LIN {X 0,Y 247.028,Z 622.984,A -85,B 0,C 180,E1 -18810.001,E2 -18810.001} C_VEL
LIN {X 0,Y 246.912,Z 622.365,A -85,B 0,C 180,E1 -18813.264,E2 -18813.264} C_VEL
LIN {X 0,Y 246.95,Z 620.585,A -85,B 0,C 180,E1 -18816.537,E2 -18816.537} C_VEL
LIN {X 0,Y 247.222,Z 617.621,A -85,B 0,C 180,E1 -18819.822,E2 -18819.822} C_VEL
LIN {X 0,Y 248.048,Z 613.414,A -85,B 0,C 180,E1 -18823.102,E2 -18823.102} C_VEL
LIN {X 0,Y 249.417,Z 607.853,A -85,B 0,C 180,E1 -18826.367,E2 -18826.367} C_VEL
LIN {X 0,Y 251.498,Z 600.794,A -85,B 0,C 180,E1 -18829.594,E2 -18829.594} C_VEL
LIN {X 0,Y 253.864,Z 593.254,A -85,B 0,C 180,E1 -18832.375,E2 -18832.375} C_VEL
LIN {X 0,Y 256.688,Z 584.514,A -85,B 0,C 180,E1 -18835.005,E2 -18835.005} C_VEL
LIN {X 0,Y 259.73,Z 574.915,A -85,B 0,C 180,E1 -18837.388,E2 -18837.388} C_VEL
LIN {X 0,Y 263.123,Z 564.018,A -85,B 0,C 180,E1 -18839.614,E2 -18839.614} C_VEL
LIN {X 0,Y 266.592,Z 552.132,A -85,B 0,C 180,E1 -18841.599,E2 -18841.599} C_VEL
LIN {X 0,Y 270.114,Z 539.053,A -85,B 0,C 180,E1 -18843.357,E2 -18843.357} C_VEL
LIN {X 0,Y 273.369,Z 524.786,A -85,B 0,C 180,E1 -18844.892,E2 -18844.892} C_VEL
LIN {X 0,Y 276.063,Z 510.769,A -85,B 0,C 180,E1 -18846.067,E2 -18846.067} C_VEL
LIN {X 0,Y 278.527,Z 495.775,A -85,B 0,C 180,E1 -18846.989,E2 -18846.989} C_VEL
LIN {X 0,Y 280.288,Z 480.084,A -85,B 0,C 180,E1 -18847.676,E2 -18847.676} C_VEL
LIN {X 0,Y 281.51,Z 460.198,A -85,B 0,C 180,E1 -18848.22,E2 -18848.22} C_VEL
LIN {X 0,Y 285.491,Z 375.925,A -85,B 0,C 180,E1 -18850.259,E2 -18850.259} C_VEL
LIN {X 0,Y 284.689,Z 371.253,A -85,B 0,C 180,E1 -18850.546,E2 -18850.546} C_VEL
LIN {X 0,Y 277.977,Z 355.557,A -85,B 0,C 180,E1 -18852.259,E2 -18852.259} C_VEL
LIN {X 0,Y 269.371,Z 338.427,A -85,B 0,C 180,E1 -18854.55,E2 -18854.55} C_VEL
LIN {X 0,Y 262.911,Z 327.193,A -85,B 0,C 180,E1 -18856.37,E2 -18856.37} C_VEL
LIN {X 0,Y 257.461,Z 318.292,A -85,B 0,C 180,E1 -18858.004,E2 -18858.004} C_VEL
LIN {X 0,Y 253.878,Z 312.814,A -85,B 0,C 180,E1 -18859.131,E2 -18859.131} C_VEL
LIN {X 0,Y 251.04,Z 308.21,A -85,B 0,C 180,E1 -18860.113,E2 -18860.113} C_VEL
LIN {X 0,Y 249.08,Z 302.081,A -85,B 0,C 180,E1 -18863.167,E2 -18863.167} C_VEL
LIN {X 0,Y 249.036,Z 302.078,A -85,B 0,C 180,E1 -18867.848,E2 -18867.848} C_VEL
LIN {X 0,Y 249.053,Z 302.077,A -85,B 0,C 180,E1 -18871.333,E2 -18871.333} C_VEL
LIN {X 0,Y 249.106,Z 302.075,A -85,B 0,C 180,E1 -18874.964,E2 -18874.964} C_VEL
LIN {X 0,Y 249.097,Z 302.078,A -85,B 0,C 180,E1 -18878.603,E2 -18878.603} C_VEL
LIN {X 0,Y 249.247,Z 302.059,A -85,B 0,C 180,E1 -18883.622,E2 -18883.622} C_VEL
LIN {X 0,Y 249.248,Z 302.052,A -85,B 0,C 180,E1 -18888.617,E2 -18888.617} C_VEL
LIN {X 0,Y 249.422,Z 302.034,A -85,B 0,C 180,E1 -18891.901,E2 -18891.901} C_VEL
LIN {X 0,Y 249.268,Z 302.06,A -85,B 0,C 180,E1 -18895.148,E2 -18895.148} C_VEL
LIN {X 0,Y 249.665,Z 302.005,A -85,B 0,C 180,E1 -18898.387,E2 -18898.387} C_VEL
LIN {X 0,Y 249.664,Z 302,A -85,B 0,C 180,E1 -18901.613,E2 -18901.613} C_VEL
LIN {X 0,Y 249.429,Z 302.029,A -85,B 0,C 180,E1 -18906.55,E2 -18906.55} C_VEL
LIN {X 0,Y 249.337,Z 302.042,A -85,B 0,C 180,E1 -18909.737,E2 -18909.737} C_VEL
LIN {X 0,Y 249.154,Z 302.063,A -85,B 0,C 180,E1 -18914.707,E2 -18914.707} C_VEL
LIN {X 0,Y 249.083,Z 302.076,A -85,B 0,C 180,E1 -18918.082,E2 -18918.082} C_VEL
LIN {X 0,Y 249.047,Z 302.084,A -85,B 0,C 180,E1 -18921.522,E2 -18921.522} C_VEL
LIN {X 0,Y 249.048,Z 302.082,A -85,B 0,C 180,E1 -18925.44,E2 -18925.44} C_VEL
LIN {X 0,Y 249.027,Z 302.058,A -85,B 0,C 180,E1 -18928.968,E2 -18928.968} C_VEL
LIN {X 0,Y 249.03,Z 302.085,A -85,B 0,C 180,E1 -18932.426,E2 -18932.426} C_VEL
LIN {X 0,Y 249.017,Z 302.084,A -85,B 0,C 180,E1 -18936.348,E2 -18936.348} C_VEL
LIN {X 0,Y 249.008,Z 302.088,A -85,B 0,C 180,E1 -18939.667,E2 -18939.667} C_VEL
LIN {X 0,Y 249.883,Z 304.763,A -85,B 0,C 180,E1 -18940.038,E2 -18940.038} C_VEL
LIN {X 0,Y 251.945,Z 307.034,A -85,B 0,C 180,E1 -18940.696,E2 -18940.696} C_VEL
LIN {X 0,Y 252.595,Z 307.715,A -85,B 0,C 180,E1 -18940.898,E2 -18940.898} C_VEL
LIN {X 0,Y 254.606,Z 310.9,A -85,B 0,C 180,E1 -18941.557,E2 -18941.557} C_VEL
LIN {X 0,Y 256.287,Z 312.966,A -85,B 0,C 180,E1 -18942.069,E2 -18942.069} C_VEL
LIN {X 0,Y 263.057,Z 322.542,A -85,B 0,C 180,E1 -18944.065,E2 -18944.065} C_VEL
LIN {X 0,Y 271.703,Z 335.608,A -85,B 0,C 180,E1 -18946.408,E2 -18946.408} C_VEL
LIN {X 0,Y 279.499,Z 348.777,A -85,B 0,C 180,E1 -18948.373,E2 -18948.373} C_VEL
LIN {X 0,Y 285.118,Z 360.529,A -85,B 0,C 180,E1 -18949.761,E2 -18949.761} C_VEL
LIN {X 0,Y 285.903,Z 362.245,A -85,B 0,C 180,E1 -18949.951,E2 -18949.951} C_VEL
LIN {X 0,Y 283.998,Z 405.185,A -85,B 0,C 180,E1 -18951.012,E2 -18951.012} C_VEL
LIN {X 0,Y 281.278,Z 459.949,A -85,B 0,C 180,E1 -18952.366,E2 -18952.366} C_VEL
LIN {X 0,Y 279.82,Z 475.194,A -85,B 0,C 180,E1 -18952.991,E2 -18952.991} C_VEL
LIN {X 0,Y 277.811,Z 490.445,A -85,B 0,C 180,E1 -18953.916,E2 -18953.916} C_VEL
LIN {X 0,Y 275.351,Z 505.031,A -85,B 0,C 180,E1 -18955.111,E2 -18955.111} C_VEL
LIN {X 0,Y 272.494,Z 518.739,A -85,B 0,C 180,E1 -18956.543,E2 -18956.543} C_VEL
LIN {X 0,Y 269.166,Z 532.173,A -85,B 0,C 180,E1 -18958.299,E2 -18958.299} C_VEL
LIN {X 0,Y 265.645,Z 544.366,A -85,B 0,C 180,E1 -18960.26,E2 -18960.26} C_VEL
LIN {X 0,Y 262.454,Z 555.296,A -85,B 0,C 180,E1 -18962.447,E2 -18962.447} C_VEL
LIN {X 0,Y 258.879,Z 566.228,A -85,B 0,C 180,E1 -18965.115,E2 -18965.115} C_VEL
LIN {X 0,Y 255.837,Z 575.164,A -85,B 0,C 180,E1 -18967.807,E2 -18967.807} C_VEL
LIN {X 0,Y 253.075,Z 583.119,A -85,B 0,C 180,E1 -18970.769,E2 -18970.769} C_VEL
LIN {X 0,Y 251.07,Z 589.468,A -85,B 0,C 180,E1 -18973.744,E2 -18973.744} C_VEL
LIN {X 0,Y 249.279,Z 594.892,A -85,B 0,C 180,E1 -18976.964,E2 -18976.964} C_VEL
LIN {X 0,Y 248.13,Z 598.978,A -85,B 0,C 180,E1 -18980.215,E2 -18980.215} C_VEL
LIN {X 0,Y 247.428,Z 602.061,A -85,B 0,C 180,E1 -18983.8,E2 -18983.8} C_VEL
LIN {X 0,Y 247.152,Z 603.561,A -85,B 0,C 180,E1 -18986.739,E2 -18986.739} C_VEL
LIN {X 0,Y 247.038,Z 604.161,A -85,B 0,C 180,E1 -18989.999,E2 -18989.999} C_VEL
LIN {X 0,Y 247.152,Z 603.6,A -85,B 0,C 180,E1 -18993.26,E2 -18993.26} C_VEL
LIN {X 0,Y 247.466,Z 601.933,A -85,B 0,C 180,E1 -18996.522,E2 -18996.522} C_VEL
LIN {X 0,Y 248.124,Z 599.116,A -85,B 0,C 180,E1 -18999.784,E2 -18999.784} C_VEL
LIN {X 0,Y 249.243,Z 595.078,A -85,B 0,C 180,E1 -19003.036,E2 -19003.036} C_VEL
LIN {X 0,Y 250.981,Z 589.715,A -85,B 0,C 180,E1 -19006.261,E2 -19006.261} C_VEL
LIN {X 0,Y 253.197,Z 582.877,A -85,B 0,C 180,E1 -19009.455,E2 -19009.455} C_VEL
LIN {X 0,Y 256.148,Z 574.329,A -85,B 0,C 180,E1 -19012.588,E2 -19012.588} C_VEL
LIN {X 0,Y 259.241,Z 565.234,A -85,B 0,C 180,E1 -19015.275,E2 -19015.275} C_VEL
LIN {X 0,Y 262.588,Z 554.812,A -85,B 0,C 180,E1 -19017.787,E2 -19017.787} C_VEL
LIN {X 0,Y 266.143,Z 542.902,A -85,B 0,C 180,E1 -19020.114,E2 -19020.114} C_VEL
LIN {X 0,Y 269.646,Z 530.412,A -85,B 0,C 180,E1 -19022.076,E2 -19022.076} C_VEL
LIN {X 0,Y 272.729,Z 518.137,A -85,B 0,C 180,E1 -19023.644,E2 -19023.644} C_VEL
LIN {X 0,Y 275.411,Z 504.945,A -85,B 0,C 180,E1 -19025.024,E2 -19025.024} C_VEL
LIN {X 0,Y 277.966,Z 490.071,A -85,B 0,C 180,E1 -19026.228,E2 -19026.228} C_VEL
LIN {X 0,Y 279.996,Z 474.56,A -85,B 0,C 180,E1 -19027.155,E2 -19027.155} C_VEL
LIN {X 0,Y 281.417,Z 459.114,A -85,B 0,C 180,E1 -19027.78,E2 -19027.78} C_VEL
LIN {X 0,Y 286.065,Z 363.468,A -85,B 0,C 180,E1 -19030.117,E2 -19030.117} C_VEL
LIN {X 0,Y 285.824,Z 361.933,A -85,B 0,C 180,E1 -19030.207,E2 -19030.207} C_VEL
LIN {X 0,Y 279.964,Z 349.532,A -85,B 0,C 180,E1 -19031.655,E2 -19031.655} C_VEL
LIN {X 0,Y 271.73,Z 335.573,A -85,B 0,C 180,E1 -19033.732,E2 -19033.732} C_VEL
LIN {X 0,Y 263.143,Z 322.632,A -85,B 0,C 180,E1 -19036.064,E2 -19036.064} C_VEL
LIN {X 0,Y 258.197,Z 315.646,A -85,B 0,C 180,E1 -19037.507,E2 -19037.507} C_VEL
LIN {X 0,Y 255.336,Z 311.626,A -85,B 0,C 180,E1 -19038.386,E2 -19038.386} C_VEL
LIN {X 0,Y 253.016,Z 308.534,A -85,B 0,C 180,E1 -19039.118,E2 -19039.118} C_VEL
LIN {X 0,Y 252.279,Z 307.253,A -85,B 0,C 180,E1 -19039.369,E2 -19039.369} C_VEL
LIN {X 0,Y 250.179,Z 305.258,A -85,B 0,C 180,E1 -19040.025,E2 -19040.025} C_VEL
LIN {X 0,Y 249.085,Z 302.629,A -85,B 0,C 180,E1 -19040.446,E2 -19040.446} C_VEL
LIN {X 0,Y 248.988,Z 302.096,A -85,B 0,C 180,E1 -19040.573,E2 -19040.573} C_VEL
LIN {X 0,Y 249.04,Z 302.058,A -85,B 0,C 180,E1 -19044.923,E2 -19044.923} C_VEL
LIN {X 0,Y 249.029,Z 302.085,A -85,B 0,C 180,E1 -19047.848,E2 -19047.848} C_VEL
LIN {X 0,Y 249.032,Z 302.087,A -85,B 0,C 180,E1 -19051.33,E2 -19051.33} C_VEL
LIN {X 0,Y 249.053,Z 302.087,A -85,B 0,C 180,E1 -19054.958,E2 -19054.958} C_VEL
LIN {X 0,Y 249.048,Z 302.088,A -85,B 0,C 180,E1 -19058.627,E2 -19058.627} C_VEL
LIN {X 0,Y 249.033,Z 302.078,A -85,B 0,C 180,E1 -19060.387,E2 -19060.387} C_VEL
LIN {X 0,Y 248.35,Z 302.163,A -85,B 0,C 180,E1 -19061.738,E2 -19061.738} C_VEL
LIN {X 0,Y 245.524,Z 302.527,A -85,B 0,C 180,E1 -19063.943,E2 -19063.943} C_VEL
LIN {X 0,Y 243.161,Z 302.812,A -85,B 0,C 180,E1 -19065.738,E2 -19065.738} C_VEL
LIN {X 0,Y 242.18,Z 302.934,A -85,B 0,C 180,E1 -19067.13,E2 -19067.13} C_VEL
LIN {X 0,Y 242.116,Z 302.943,A -85,B 0,C 180,E1 -19067.601,E2 -19067.601} C_VEL
LIN {X 0,Y 242.369,Z 302.906,A -85,B 0,C 180,E1 -19071.663,E2 -19071.663} C_VEL
LIN {X 0,Y 242.395,Z 302.917,A -85,B 0,C 180,E1 -19073.34,E2 -19073.34} C_VEL
LIN {X 0,Y 242.619,Z 302.89,A -85,B 0,C 180,E1 -19078.34,E2 -19078.34} C_VEL
LIN {X 0,Y 242.62,Z 302.873,A -85,B 0,C 180,E1 -19081.66,E2 -19081.66} C_VEL
LIN {X 0,Y 242.4,Z 302.902,A -85,B 0,C 180,E1 -19086.66,E2 -19086.66} C_VEL
LIN {X 0,Y 242.265,Z 302.92,A -85,B 0,C 180,E1 -19090.024,E2 -19090.024} C_VEL
LIN {X 0,Y 242.165,Z 302.933,A -85,B 0,C 180,E1 -19095.141,E2 -19095.141} C_VEL
LIN {X 0,Y 242.077,Z 302.949,A -85,B 0,C 180,E1 -19098.624,E2 -19098.624} C_VEL
LIN {X 0,Y 242.039,Z 302.959,A -85,B 0,C 180,E1 -19102.177,E2 -19102.177} C_VEL
LIN {X 0,Y 242.03,Z 302.921,A -85,B 0,C 180,E1 -19105.821,E2 -19105.821} C_VEL
LIN {X 0,Y 241.967,Z 302.96,A -85,B 0,C 180,E1 -19109.588,E2 -19109.588} C_VEL
LIN {X 0,Y 241.977,Z 302.944,A -85,B 0,C 180,E1 -19113.493,E2 -19113.493} C_VEL
LIN {X 0,Y 242.013,Z 302.997,A -85,B 0,C 180,E1 -19115.124,E2 -19115.124} C_VEL
LIN {X 0,Y 243.78,Z 308.093,A -85,B 0,C 180,E1 -19117.771,E2 -19117.771} C_VEL
LIN {X 0,Y 247.145,Z 313.192,A -85,B 0,C 180,E1 -19118.988,E2 -19118.988} C_VEL
LIN {X 0,Y 252.342,Z 321.207,A -85,B 0,C 180,E1 -19120.754,E2 -19120.754} C_VEL
LIN {X 0,Y 258.208,Z 330.752,A -85,B 0,C 180,E1 -19122.613,E2 -19122.613} C_VEL
LIN {X 0,Y 265.538,Z 343.696,A -85,B 0,C 180,E1 -19124.778,E2 -19124.778} C_VEL
LIN {X 0,Y 273.318,Z 359.407,A -85,B 0,C 180,E1 -19126.939,E2 -19126.939} C_VEL
LIN {X 0,Y 279.864,Z 374.827,A -85,B 0,C 180,E1 -19128.685,E2 -19128.685} C_VEL
LIN {X 0,Y 280.063,Z 378.719,A -85,B 0,C 180,E1 -19128.85,E2 -19128.85} C_VEL
LIN {X 0,Y 275.26,Z 474.583,A -85,B 0,C 180,E1 -19131.22,E2 -19131.22} C_VEL
LIN {X 0,Y 273.789,Z 489.624,A -85,B 0,C 180,E1 -19131.796,E2 -19131.796} C_VEL
LIN {X 0,Y 271.499,Z 505.04,A -85,B 0,C 180,E1 -19132.649,E2 -19132.649} C_VEL
LIN {X 0,Y 268.772,Z 519.31,A -85,B 0,C 180,E1 -19133.729,E2 -19133.729} C_VEL
LIN {X 0,Y 265.63,Z 533.215,A -85,B 0,C 180,E1 -19135.104,E2 -19135.104} C_VEL
LIN {X 0,Y 262.333,Z 545.919,A -85,B 0,C 180,E1 -19136.688,E2 -19136.688} C_VEL
LIN {X 0,Y 258.552,Z 558.802,A -85,B 0,C 180,E1 -19138.678,E2 -19138.678} C_VEL
LIN {X 0,Y 255.103,Z 569.595,A -85,B 0,C 180,E1 -19140.726,E2 -19140.726} C_VEL
LIN {X 0,Y 251.818,Z 579.592,A -85,B 0,C 180,E1 -19143.031,E2 -19143.031} C_VEL
LIN {X 0,Y 248.578,Z 589.386,A -85,B 0,C 180,E1 -19145.799,E2 -19145.799} C_VEL
LIN {X 0,Y 245.766,Z 597.563,A -85,B 0,C 180,E1 -19148.618,E2 -19148.618} C_VEL
LIN {X 0,Y 243.527,Z 604.333,A -85,B 0,C 180,E1 -19151.492,E2 -19151.492} C_VEL
LIN {X 0,Y 241.716,Z 610.597,A -85,B 0,C 180,E1 -19154.831,E2 -19154.831} C_VEL
LIN {X 0,Y 240.513,Z 615.451,A -85,B 0,C 180,E1 -19158.198,E2 -19158.198} C_VEL
LIN {X 0,Y 239.943,Z 619.017,A -85,B 0,C 180,E1 -19161.579,E2 -19161.579} C_VEL
LIN {X 0,Y 239.837,Z 621.429,A -85,B 0,C 180,E1 -19165.074,E2 -19165.074} C_VEL
LIN {X 0,Y 239.888,Z 622.557,A -85,B 0,C 180,E1 -19168.322,E2 -19168.322} C_VEL
LIN {X 0,Y 239.957,Z 622.715,A -85,B 0,C 180,E1 -19170.001,E2 -19170.001} C_VEL
LIN {X 0,Y 239.815,Z 622.094,A -85,B 0,C 180,E1 -19173.361,E2 -19173.361} C_VEL
LIN {X 0,Y 239.866,Z 620.313,A -85,B 0,C 180,E1 -19176.731,E2 -19176.731} C_VEL
LIN {X 0,Y 240.158,Z 617.347,A -85,B 0,C 180,E1 -19180.114,E2 -19180.114} C_VEL
LIN {X 0,Y 241.068,Z 613.14,A -85,B 0,C 180,E1 -19183.488,E2 -19183.488} C_VEL
LIN {X 0,Y 242.522,Z 607.577,A -85,B 0,C 180,E1 -19186.846,E2 -19186.846} C_VEL
LIN {X 0,Y 244.739,Z 600.519,A -85,B 0,C 180,E1 -19190.158,E2 -19190.158} C_VEL
LIN {X 0,Y 247.268,Z 592.98,A -85,B 0,C 180,E1 -19193.006,E2 -19193.006} C_VEL
LIN {X 0,Y 250.189,Z 584.278,A -85,B 0,C 180,E1 -19195.688,E2 -19195.688} C_VEL
LIN {X 0,Y 253.369,Z 574.639,A -85,B 0,C 180,E1 -19198.136,E2 -19198.136} C_VEL
LIN {X 0,Y 256.922,Z 563.742,A -85,B 0,C 180,E1 -19200.403,E2 -19200.403} C_VEL
LIN {X 0,Y 260.554,Z 551.857,A -85,B 0,C 180,E1 -19202.419,E2 -19202.419} C_VEL
LIN {X 0,Y 264.069,Z 539.239,A -85,B 0,C 180,E1 -19204.151,E2 -19204.151} C_VEL
LIN {X 0,Y 267.173,Z 526.281,A -85,B 0,C 180,E1 -19205.592,E2 -19205.592} C_VEL
LIN {X 0,Y 270.132,Z 511.621,A -85,B 0,C 180,E1 -19206.872,E2 -19206.872} C_VEL
LIN {X 0,Y 272.784,Z 496.259,A -85,B 0,C 180,E1 -19207.844,E2 -19207.844} C_VEL
LIN {X 0,Y 274.588,Z 480.943,A -85,B 0,C 180,E1 -19208.542,E2 -19208.542} C_VEL
LIN {X 0,Y 275.885,Z 461.698,A -85,B 0,C 180,E1 -19209.087,E2 -19209.087} C_VEL
LIN {X 0,Y 280.043,Z 377.146,A -85,B 0,C 180,E1 -19211.159,E2 -19211.159} C_VEL
LIN {X 0,Y 279.467,Z 374.025,A -85,B 0,C 180,E1 -19211.366,E2 -19211.366} C_VEL
LIN {X 0,Y 272.793,Z 358.422,A -85,B 0,C 180,E1 -19213.146,E2 -19213.146} C_VEL
LIN {X 0,Y 265.042,Z 342.882,A -85,B 0,C 180,E1 -19215.301,E2 -19215.301} C_VEL
LIN {X 0,Y 258.725,Z 331.72,A -85,B 0,C 180,E1 -19217.161,E2 -19217.161} C_VEL
LIN {X 0,Y 253.359,Z 322.874,A -85,B 0,C 180,E1 -19218.842,E2 -19218.842} C_VEL
LIN {X 0,Y 249.941,Z 317.542,A -85,B 0,C 180,E1 -19219.968,E2 -19219.968} C_VEL
LIN {X 0,Y 246.621,Z 312.568,A -85,B 0,C 180,E1 -19221.11,E2 -19221.11} C_VEL
LIN {X 0,Y 243.599,Z 307.701,A -85,B 0,C 180,E1 -19222.28,E2 -19222.28} C_VEL
LIN {X 0,Y 242.001,Z 302.956,A -85,B 0,C 180,E1 -19224.874,E2 -19224.874} C_VEL
LIN {X 0,Y 241.956,Z 302.963,A -85,B 0,C 180,E1 -19228.477,E2 -19228.477} C_VEL
LIN {X 0,Y 241.972,Z 302.965,A -85,B 0,C 180,E1 -19232.308,E2 -19232.308} C_VEL
LIN {X 0,Y 242.03,Z 302.957,A -85,B 0,C 180,E1 -19236.013,E2 -19236.013} C_VEL
LIN {X 0,Y 242.04,Z 302.958,A -85,B 0,C 180,E1 -19239.608,E2 -19239.608} C_VEL
LIN {X 0,Y 242.168,Z 302.945,A -85,B 0,C 180,E1 -19243.279,E2 -19243.279} C_VEL
LIN {X 0,Y 242.185,Z 302.932,A -85,B 0,C 180,E1 -19248.28,E2 -19248.28} C_VEL
LIN {X 0,Y 242.376,Z 302.914,A -85,B 0,C 180,E1 -19251.664,E2 -19251.664} C_VEL
LIN {X 0,Y 242.401,Z 302.904,A -85,B 0,C 180,E1 -19253.34,E2 -19253.34} C_VEL
LIN {X 0,Y 242.625,Z 302.881,A -85,B 0,C 180,E1 -19258.34,E2 -19258.34} C_VEL
LIN {X 0,Y 242.624,Z 302.876,A -85,B 0,C 180,E1 -19261.66,E2 -19261.66} C_VEL
LIN {X 0,Y 242.405,Z 302.904,A -85,B 0,C 180,E1 -19266.66,E2 -19266.66} C_VEL
LIN {X 0,Y 242.265,Z 302.921,A -85,B 0,C 180,E1 -19270.024,E2 -19270.024} C_VEL
LIN {X 0,Y 242.111,Z 302.94,A -85,B 0,C 180,E1 -19275.145,E2 -19275.145} C_VEL
LIN {X 0,Y 242.021,Z 302.952,A -85,B 0,C 180,E1 -19278.628,E2 -19278.628} C_VEL
LIN {X 0,Y 241.977,Z 302.96,A -85,B 0,C 180,E1 -19282.184,E2 -19282.184} C_VEL
LIN {X 0,Y 241.99,Z 302.954,A -85,B 0,C 180,E1 -19285.826,E2 -19285.826} C_VEL
LIN {X 0,Y 241.966,Z 302.943,A -85,B 0,C 180,E1 -19289.589,E2 -19289.589} C_VEL
LIN {X 0,Y 241.982,Z 302.962,A -85,B 0,C 180,E1 -19293.493,E2 -19293.493} C_VEL
LIN {X 0,Y 242.01,Z 303.038,A -85,B 0,C 180,E1 -19297.657,E2 -19297.657} C_VEL
LIN {X 0,Y 242.888,Z 305.613,A -85,B 0,C 180,E1 -19298.05,E2 -19298.05} C_VEL
LIN {X 0,Y 244.943,Z 307.902,A -85,B 0,C 180,E1 -19298.772,E2 -19298.772} C_VEL
LIN {X 0,Y 245.748,Z 308.748,A -85,B 0,C 180,E1 -19299.046,E2 -19299.046} C_VEL
LIN {X 0,Y 247.873,Z 312.052,A -85,B 0,C 180,E1 -19299.802,E2 -19299.802} C_VEL
LIN {X 0,Y 249.338,Z 313.637,A -85,B 0,C 180,E1 -19300.278,E2 -19300.278} C_VEL
LIN {X 0,Y 252.02,Z 317.353,A -85,B 0,C 180,E1 -19301.158,E2 -19301.158} C_VEL
LIN {X 0,Y 259.541,Z 328.105,A -85,B 0,C 180,E1 -19303.47,E2 -19303.47} C_VEL
LIN {X 0,Y 267.969,Z 341.061,A -85,B 0,C 180,E1 -19305.836,E2 -19305.836} C_VEL
LIN {X 0,Y 275.738,Z 354.452,A -85,B 0,C 180,E1 -19307.863,E2 -19307.863} C_VEL
LIN {X 0,Y 280.38,Z 364.54,A -85,B 0,C 180,E1 -19309.062,E2 -19309.062} C_VEL
LIN {X 0,Y 278.6,Z 404.339,A -85,B 0,C 180,E1 -19310.07,E2 -19310.07} C_VEL
LIN {X 0,Y 275.708,Z 460.234,A -85,B 0,C 180,E1 -19311.469,E2 -19311.469} C_VEL
LIN {X 0,Y 274.216,Z 475.392,A -85,B 0,C 180,E1 -19312.098,E2 -19312.098} C_VEL
LIN {X 0,Y 272.229,Z 490.12,A -85,B 0,C 180,E1 -19312.997,E2 -19312.997} C_VEL
LIN {X 0,Y 269.768,Z 504.15,A -85,B 0,C 180,E1 -19314.139,E2 -19314.139} C_VEL
LIN {X 0,Y 266.611,Z 519.014,A -85,B 0,C 180,E1 -19315.704,E2 -19315.704} C_VEL
LIN {X 0,Y 263.147,Z 532.448,A -85,B 0,C 180,E1 -19317.486,E2 -19317.486} C_VEL
LIN {X 0,Y 259.483,Z 544.64,A -85,B 0,C 180,E1 -19319.479,E2 -19319.479} C_VEL
LIN {X 0,Y 256.075,Z 555.824,A -85,B 0,C 180,E1 -19321.766,E2 -19321.766} C_VEL
LIN {X 0,Y 252.409,Z 566.503,A -85,B 0,C 180,E1 -19324.431,E2 -19324.431} C_VEL
LIN {X 0,Y 249.258,Z 575.438,A -85,B 0,C 180,E1 -19327.188,E2 -19327.188} C_VEL
LIN {X 0,Y 246.258,Z 583.699,A -85,B 0,C 180,E1 -19330.355,E2 -19330.355} C_VEL
LIN {X 0,Y 244.221,Z 589.741,A -85,B 0,C 180,E1 -19333.275,E2 -19333.275} C_VEL
LIN {X 0,Y 242.334,Z 595.165,A -85,B 0,C 180,E1 -19336.584,E2 -19336.584} C_VEL
LIN {X 0,Y 241.115,Z 599.25,A -85,B 0,C 180,E1 -19339.927,E2 -19339.927} C_VEL
LIN {X 0,Y 240.327,Z 602.498,A -85,B 0,C 180,E1 -19343.87,E2 -19343.87} C_VEL
LIN {X 0,Y 240.072,Z 603.832,A -85,B 0,C 180,E1 -19346.643,E2 -19346.643} C_VEL
LIN {X 0,Y 239.968,Z 604.431,A -85,B 0,C 180,E1 -19349.999,E2 -19349.999} C_VEL
LIN {X 0,Y 240.071,Z 603.87,A -85,B 0,C 180,E1 -19353.356,E2 -19353.356} C_VEL
LIN {X 0,Y 240.405,Z 602.203,A -85,B 0,C 180,E1 -19356.715,E2 -19356.715} C_VEL
LIN {X 0,Y 241.106,Z 599.387,A -85,B 0,C 180,E1 -19360.072,E2 -19360.072} C_VEL
LIN {X 0,Y 242.298,Z 595.349,A -85,B 0,C 180,E1 -19363.417,E2 -19363.417} C_VEL
LIN {X 0,Y 244.139,Z 589.985,A -85,B 0,C 180,E1 -19366.73,E2 -19366.73} C_VEL
LIN {X 0,Y 246.501,Z 583.147,A -85,B 0,C 180,E1 -19370.006,E2 -19370.006} C_VEL
LIN {X 0,Y 249.579,Z 574.599,A -85,B 0,C 180,E1 -19373.217,E2 -19373.217} C_VEL
LIN {X 0,Y 252.799,Z 565.503,A -85,B 0,C 180,E1 -19375.967,E2 -19375.967} C_VEL
LIN {X 0,Y 256.162,Z 555.564,A -85,B 0,C 180,E1 -19378.424,E2 -19378.424} C_VEL
LIN {X 0,Y 260.04,Z 543.168,A -85,B 0,C 180,E1 -19380.897,E2 -19380.897} C_VEL
LIN {X 0,Y 263.645,Z 530.679,A -85,B 0,C 180,E1 -19382.897,E2 -19382.897} C_VEL
LIN {X 0,Y 266.857,Z 518.401,A -85,B 0,C 180,E1 -19384.487,E2 -19384.487} C_VEL
LIN {X 0,Y 269.519,Z 505.784,A -85,B 0,C 180,E1 -19385.832,E2 -19385.832} C_VEL
LIN {X 0,Y 272.107,Z 491.479,A -85,B 0,C 180,E1 -19387.021,E2 -19387.021} C_VEL
LIN {X 0,Y 274.289,Z 475.663,A -85,B 0,C 180,E1 -19388.005,E2 -19388.005} C_VEL
LIN {X 0,Y 275.744,Z 460.643,A -85,B 0,C 180,E1 -19388.641,E2 -19388.641} C_VEL
LIN {X 0,Y 278.922,Z 400.431,A -85,B 0,C 180,E1 -19390.14,E2 -19390.14} C_VEL
LIN {X 0,Y 280.554,Z 364.78,A -85,B 0,C 180,E1 -19391.036,E2 -19391.036} C_VEL
LIN {X 0,Y 275.21,Z 353.452,A -85,B 0,C 180,E1 -19392.413,E2 -19392.413} C_VEL
LIN {X 0,Y 267.523,Z 340.302,A -85,B 0,C 180,E1 -19394.433,E2 -19394.433} C_VEL
LIN {X 0,Y 259.654,Z 328.232,A -85,B 0,C 180,E1 -19396.653,E2 -19396.653} C_VEL
LIN {X 0,Y 254.38,Z 320.716,A -85,B 0,C 180,E1 -19398.251,E2 -19398.251} C_VEL
LIN {X 0,Y 251.667,Z 316.899,A -85,B 0,C 180,E1 -19399.117,E2 -19399.117} C_VEL
LIN {X 0,Y 248.629,Z 312.791,A -85,B 0,C 180,E1 -19400.122,E2 -19400.122} C_VEL
LIN {X 0,Y 246.245,Z 309.779,A -85,B 0,C 180,E1 -19400.933,E2 -19400.933} C_VEL
LIN {X 0,Y 245.457,Z 308.214,A -85,B 0,C 180,E1 -19401.234,E2 -19401.234} C_VEL
LIN {X 0,Y 243.346,Z 306.328,A -85,B 0,C 180,E1 -19401.952,E2 -19401.952} C_VEL
LIN {X 0,Y 242.195,Z 303.988,A -85,B 0,C 180,E1 -19402.416,E2 -19402.416} C_VEL
LIN {X 0,Y 241.961,Z 302.939,A -85,B 0,C 180,E1 -19402.544,E2 -19402.544} C_VEL
LIN {X 0,Y 241.976,Z 302.966,A -85,B 0,C 180,E1 -19406.507,E2 -19406.507} C_VEL
LIN {X 0,Y 241.968,Z 302.971,A -85,B 0,C 180,E1 -19410.615,E2 -19410.615} C_VEL
LIN {X 0,Y 241.993,Z 302.965,A -85,B 0,C 180,E1 -19414.197,E2 -19414.197} C_VEL
LIN {X 0,Y 241.983,Z 302.965,A -85,B 0,C 180,E1 -19418.338,E2 -19418.338} C_VEL
LIN {X 0,Y 242.103,Z 302.953,A -85,B 0,C 180,E1 -19423.324,E2 -19423.324} C_VEL
LIN {X 0,Y 242.116,Z 302.943,A -85,B 0,C 180,E1 -19427.601,E2 -19427.601} C_VEL
LIN {X 0,Y 241.5,Z 303.031,A -85,B 0,C 180,E1 -19428.991,E2 -19428.991} C_VEL
LIN {X 0,Y 238.698,Z 303.386,A -85,B 0,C 180,E1 -19431.261,E2 -19431.261} C_VEL
LIN {X 0,Y 236.296,Z 303.678,A -85,B 0,C 180,E1 -19433.11,E2 -19433.11} C_VEL
LIN {X 0,Y 235.268,Z 303.797,A -85,B 0,C 180,E1 -19434.543,E2 -19434.543} C_VEL
LIN {X 0,Y 235.188,Z 303.801,A -85,B 0,C 180,E1 -19435.029,E2 -19435.029} C_VEL
LIN {X 0,Y 235.579,Z 303.766,A -85,B 0,C 180,E1 -19438.29,E2 -19438.29} C_VEL
LIN {X 0,Y 235.579,Z 303.75,A -85,B 0,C 180,E1 -19441.709,E2 -19441.709} C_VEL
LIN {X 0,Y 235.352,Z 303.781,A -85,B 0,C 180,E1 -19446.86,E2 -19446.86} C_VEL
LIN {X 0,Y 235.212,Z 303.797,A -85,B 0,C 180,E1 -19450.327,E2 -19450.327} C_VEL
LIN {X 0,Y 235.112,Z 303.812,A -85,B 0,C 180,E1 -19455.606,E2 -19455.606} C_VEL
LIN {X 0,Y 235.017,Z 303.826,A -85,B 0,C 180,E1 -19459.205,E2 -19459.205} C_VEL
LIN {X 0,Y 234.963,Z 303.824,A -85,B 0,C 180,E1 -19462.882,E2 -19462.882} C_VEL
LIN {X 0,Y 234.943,Z 303.81,A -85,B 0,C 180,E1 -19466.66,E2 -19466.66} C_VEL
LIN {X 0,Y 234.897,Z 303.823,A -85,B 0,C 180,E1 -19470.573,E2 -19470.573} C_VEL
LIN {X 0,Y 234.946,Z 303.861,A -85,B 0,C 180,E1 -19473.243,E2 -19473.243} C_VEL
LIN {X 0,Y 236.211,Z 307.621,A -85,B 0,C 180,E1 -19475.333,E2 -19475.333} C_VEL
LIN {X 0,Y 240.088,Z 313.151,A -85,B 0,C 180,E1 -19476.876,E2 -19476.876} C_VEL
LIN {X 0,Y 245.042,Z 320.699,A -85,B 0,C 180,E1 -19478.726,E2 -19478.726} C_VEL
LIN {X 0,Y 249.321,Z 327.378,A -85,B 0,C 180,E1 -19480.217,E2 -19480.217} C_VEL
LIN {X 0,Y 256.592,Z 339.544,A -85,B 0,C 180,E1 -19482.578,E2 -19482.578} C_VEL
LIN {X 0,Y 263.816,Z 353.172,A -85,B 0,C 180,E1 -19484.761,E2 -19484.761} C_VEL
LIN {X 0,Y 270.371,Z 367.154,A -85,B 0,C 180,E1 -19486.634,E2 -19486.634} C_VEL
LIN {X 0,Y 274.75,Z 377.81,A -85,B 0,C 180,E1 -19487.851,E2 -19487.851} C_VEL
LIN {X 0,Y 270.409,Z 462.895,A -85,B 0,C 180,E1 -19489.965,E2 -19489.965} C_VEL
LIN {X 0,Y 269.212,Z 480.453,A -85,B 0,C 180,E1 -19490.482,E2 -19490.482} C_VEL
LIN {X 0,Y 267.362,Z 495.829,A -85,B 0,C 180,E1 -19491.189,E2 -19491.189} C_VEL
LIN {X 0,Y 264.796,Z 510.677,A -85,B 0,C 180,E1 -19492.139,E2 -19492.139} C_VEL
LIN {X 0,Y 261.846,Z 524.603,A -85,B 0,C 180,E1 -19493.332,E2 -19493.332} C_VEL
LIN {X 0,Y 258.812,Z 536.989,A -85,B 0,C 180,E1 -19494.682,E2 -19494.682} C_VEL
LIN {X 0,Y 254.95,Z 550.631,A -85,B 0,C 180,E1 -19496.543,E2 -19496.543} C_VEL
LIN {X 0,Y 251.461,Z 561.696,A -85,B 0,C 180,E1 -19498.397,E2 -19498.397} C_VEL
LIN {X 0,Y 247.659,Z 572.886,A -85,B 0,C 180,E1 -19500.692,E2 -19500.692} C_VEL
LIN {X 0,Y 244.031,Z 583.418,A -85,B 0,C 180,E1 -19503.374,E2 -19503.374} C_VEL
LIN {X 0,Y 240.72,Z 592.821,A -85,B 0,C 180,E1 -19506.332,E2 -19506.332} C_VEL
LIN {X 0,Y 238.005,Z 600.347,A -85,B 0,C 180,E1 -19509.247,E2 -19509.247} C_VEL
LIN {X 0,Y 235.658,Z 607.378,A -85,B 0,C 180,E1 -19512.65,E2 -19512.65} C_VEL
LIN {X 0,Y 234.107,Z 612.921,A -85,B 0,C 180,E1 -19516.105,E2 -19516.105} C_VEL
LIN {X 0,Y 233.11,Z 617.117,A -85,B 0,C 180,E1 -19519.579,E2 -19519.579} C_VEL
LIN {X 0,Y 232.78,Z 620.072,A -85,B 0,C 180,E1 -19523.064,E2 -19523.064} C_VEL
LIN {X 0,Y 232.722,Z 621.837,A -85,B 0,C 180,E1 -19526.538,E2 -19526.538} C_VEL
LIN {X 0,Y 232.887,Z 622.445,A -85,B 0,C 180,E1 -19530.001,E2 -19530.001} C_VEL
LIN {X 0,Y 232.722,Z 621.823,A -85,B 0,C 180,E1 -19533.464,E2 -19533.464} C_VEL
LIN {X 0,Y 232.778,Z 620.041,A -85,B 0,C 180,E1 -19536.937,E2 -19536.937} C_VEL
LIN {X 0,Y 233.108,Z 617.073,A -85,B 0,C 180,E1 -19540.423,E2 -19540.423} C_VEL
LIN {X 0,Y 234.107,Z 612.866,A -85,B 0,C 180,E1 -19543.897,E2 -19543.897} C_VEL
LIN {X 0,Y 235.728,Z 607.138,A -85,B 0,C 180,E1 -19547.437,E2 -19547.437} C_VEL
LIN {X 0,Y 237.995,Z 600.243,A -85,B 0,C 180,E1 -19550.755,E2 -19550.755} C_VEL
LIN {X 0,Y 240.707,Z 592.706,A -85,B 0,C 180,E1 -19553.671,E2 -19553.671} C_VEL
LIN {X 0,Y 243.975,Z 583.387,A -85,B 0,C 180,E1 -19556.6,E2 -19556.6} C_VEL
LIN {X 0,Y 247.66,Z 572.719,A -85,B 0,C 180,E1 -19559.31,E2 -19559.31} C_VEL
LIN {X 0,Y 251.747,Z 560.471,A -85,B 0,C 180,E1 -19561.799,E2 -19561.799} C_VEL
LIN {X 0,Y 255.672,Z 547.993,A -85,B 0,C 180,E1 -19563.825,E2 -19563.825} C_VEL
LIN {X 0,Y 259.023,Z 535.785,A -85,B 0,C 180,E1 -19565.439,E2 -19565.439} C_VEL
LIN {X 0,Y 262.225,Z 522.461,A -85,B 0,C 180,E1 -19566.848,E2 -19566.848} C_VEL
LIN {X 0,Y 264.928,Z 509.084,A -85,B 0,C 180,E1 -19567.962,E2 -19567.962} C_VEL
LIN {X 0,Y 267.45,Z 494.453,A -85,B 0,C 180,E1 -19568.858,E2 -19568.858} C_VEL
LIN {X 0,Y 269.187,Z 479.516,A -85,B 0,C 180,E1 -19569.524,E2 -19569.524} C_VEL
LIN {X 0,Y 270.505,Z 459.614,A -85,B 0,C 180,E1 -19570.08,E2 -19570.08} C_VEL
LIN {X 0,Y 274.57,Z 377.554,A -85,B 0,C 180,E1 -19572.141,E2 -19572.141} C_VEL
LIN {X 0,Y 268.258,Z 362.57,A -85,B 0,C 180,E1 -19573.901,E2 -19573.901} C_VEL
LIN {X 0,Y 260.946,Z 347.638,A -85,B 0,C 180,E1 -19576.024,E2 -19576.024} C_VEL
LIN {X 0,Y 254.619,Z 336.207,A -85,B 0,C 180,E1 -19577.972,E2 -19577.972} C_VEL
LIN {X 0,Y 247.463,Z 324.307,A -85,B 0,C 180,E1 -19580.349,E2 -19580.349} C_VEL
LIN {X 0,Y 243.091,Z 317.769,A -85,B 0,C 180,E1 -19581.899,E2 -19581.899} C_VEL
LIN {X 0,Y 239.928,Z 312.962,A -85,B 0,C 180,E1 -19583.095,E2 -19583.095} C_VEL
LIN {X 0,Y 236.268,Z 307.74,A -85,B 0,C 180,E1 -19584.547,E2 -19584.547} C_VEL
LIN {X 0,Y 235.577,Z 305.926,A -85,B 0,C 180,E1 -19585.471,E2 -19585.471} C_VEL
LIN {X 0,Y 234.952,Z 303.835,A -85,B 0,C 180,E1 -19586.758,E2 -19586.758} C_VEL
LIN {X 0,Y 234.906,Z 303.839,A -85,B 0,C 180,E1 -19591.4,E2 -19591.4} C_VEL
LIN {X 0,Y 234.959,Z 303.839,A -85,B 0,C 180,E1 -19595.244,E2 -19595.244} C_VEL
LIN {X 0,Y 235.002,Z 303.837,A -85,B 0,C 180,E1 -19598.969,E2 -19598.969} C_VEL
LIN {X 0,Y 235.101,Z 303.825,A -85,B 0,C 180,E1 -19603.06,E2 -19603.06} C_VEL
LIN {X 0,Y 235.119,Z 303.815,A -85,B 0,C 180,E1 -19607.922,E2 -19607.922} C_VEL
LIN {X 0,Y 235.316,Z 303.796,A -85,B 0,C 180,E1 -19611.412,E2 -19611.412} C_VEL
LIN {X 0,Y 235.353,Z 303.781,A -85,B 0,C 180,E1 -19613.14,E2 -19613.14} C_VEL
LIN {X 0,Y 235.583,Z 303.757,A -85,B 0,C 180,E1 -19618.291,E2 -19618.291} C_VEL
LIN {X 0,Y 235.583,Z 303.753,A -85,B 0,C 180,E1 -19621.71,E2 -19621.71} C_VEL
LIN {X 0,Y 235.357,Z 303.783,A -85,B 0,C 180,E1 -19626.86,E2 -19626.86} C_VEL
LIN {X 0,Y 235.189,Z 303.802,A -85,B 0,C 180,E1 -19630.329,E2 -19630.329} C_VEL
LIN {X 0,Y 235.047,Z 303.823,A -85,B 0,C 180,E1 -19635.611,E2 -19635.611} C_VEL
LIN {X 0,Y 234.962,Z 303.832,A -85,B 0,C 180,E1 -19639.21,E2 -19639.21} C_VEL
LIN {X 0,Y 234.921,Z 303.837,A -85,B 0,C 180,E1 -19642.887,E2 -19642.887} C_VEL
LIN {X 0,Y 234.909,Z 303.821,A -85,B 0,C 180,E1 -19646.665,E2 -19646.665} C_VEL
LIN {X 0,Y 234.899,Z 303.84,A -85,B 0,C 180,E1 -19650.573,E2 -19650.573} C_VEL
LIN {X 0,Y 234.926,Z 303.847,A -85,B 0,C 180,E1 -19654.639,E2 -19654.639} C_VEL
LIN {X 0,Y 234.943,Z 303.924,A -85,B 0,C 180,E1 -19655.385,E2 -19655.385} C_VEL
LIN {X 0,Y 235.816,Z 306.503,A -85,B 0,C 180,E1 -19655.818,E2 -19655.818} C_VEL
LIN {X 0,Y 237.866,Z 308.766,A -85,B 0,C 180,E1 -19656.617,E2 -19656.617} C_VEL
LIN {X 0,Y 238.837,Z 309.514,A -85,B 0,C 180,E1 -19656.97,E2 -19656.97} C_VEL
LIN {X 0,Y 240.778,Z 312.685,A -85,B 0,C 180,E1 -19657.738,E2 -19657.738} C_VEL
LIN {X 0,Y 242.559,Z 314.597,A -85,B 0,C 180,E1 -19658.374,E2 -19658.374} C_VEL
LIN {X 0,Y 245.309,Z 318.422,A -85,B 0,C 180,E1 -19659.361,E2 -19659.361} C_VEL
LIN {X 0,Y 252.22,Z 327.975,A -85,B 0,C 180,E1 -19661.661,E2 -19661.661} C_VEL
LIN {X 0,Y 260.42,Z 340.371,A -85,B 0,C 180,E1 -19664.156,E2 -19664.156} C_VEL
LIN {X 0,Y 268.751,Z 354.251,A -85,B 0,C 180,E1 -19666.479,E2 -19666.479} C_VEL
LIN {X 0,Y 272.841,Z 362.103,A -85,B 0,C 180,E1 -19667.574,E2 -19667.574} C_VEL
LIN {X 0,Y 274.943,Z 366.872,A -85,B 0,C 180,E1 -19668.142,E2 -19668.142} C_VEL
LIN {X 0,Y 273.783,Z 393.195,A -85,B 0,C 180,E1 -19668.831,E2 -19668.831} C_VEL
LIN {X 0,Y 270.214,Z 460.52,A -85,B 0,C 180,E1 -19670.535,E2 -19670.535} C_VEL
LIN {X 0,Y 268.67,Z 475.672,A -85,B 0,C 180,E1 -19671.171,E2 -19671.171} C_VEL
LIN {X 0,Y 266.599,Z 490.398,A -85,B 0,C 180,E1 -19672.079,E2 -19672.079} C_VEL
LIN {X 0,Y 263.974,Z 504.848,A -85,B 0,C 180,E1 -19673.276,E2 -19673.276} C_VEL
LIN {X 0,Y 260.778,Z 519.289,A -85,B 0,C 180,E1 -19674.825,E2 -19674.825} C_VEL
LIN {X 0,Y 257.182,Z 532.723,A -85,B 0,C 180,E1 -19676.635,E2 -19676.635} C_VEL
LIN {X 0,Y 253.377,Z 544.915,A -85,B 0,C 180,E1 -19678.662,E2 -19678.662} C_VEL
LIN {X 0,Y 249.731,Z 556.35,A -85,B 0,C 180,E1 -19681.052,E2 -19681.052} C_VEL
LIN {X 0,Y 246.006,Z 566.777,A -85,B 0,C 180,E1 -19683.716,E2 -19683.716} C_VEL
LIN {X 0,Y 242.698,Z 575.711,A -85,B 0,C 180,E1 -19686.535,E2 -19686.535} C_VEL
LIN {X 0,Y 239.855,Z 583.111,A -85,B 0,C 180,E1 -19689.413,E2 -19689.413} C_VEL
LIN {X 0,Y 237.397,Z 590.015,A -85,B 0,C 180,E1 -19692.779,E2 -19692.779} C_VEL
LIN {X 0,Y 235.41,Z 595.438,A -85,B 0,C 180,E1 -19696.181,E2 -19696.181} C_VEL
LIN {X 0,Y 234.117,Z 599.521,A -85,B 0,C 180,E1 -19699.623,E2 -19699.623} C_VEL
LIN {X 0,Y 233.362,Z 602.384,A -85,B 0,C 180,E1 -19703.08,E2 -19703.08} C_VEL
LIN {X 0,Y 232.993,Z 604.102,A -85,B 0,C 180,E1 -19706.541,E2 -19706.541} C_VEL
LIN {X 0,Y 232.899,Z 604.7,A -85,B 0,C 180,E1 -19709.999,E2 -19709.999} C_VEL
LIN {X 0,Y 232.993,Z 604.14,A -85,B 0,C 180,E1 -19713.458,E2 -19713.458} C_VEL
LIN {X 0,Y 233.361,Z 602.473,A -85,B 0,C 180,E1 -19716.918,E2 -19716.918} C_VEL
LIN {X 0,Y 234.107,Z 599.657,A -85,B 0,C 180,E1 -19720.376,E2 -19720.376} C_VEL
LIN {X 0,Y 235.375,Z 595.619,A -85,B 0,C 180,E1 -19723.819,E2 -19723.819} C_VEL
LIN {X 0,Y 237.319,Z 590.255,A -85,B 0,C 180,E1 -19727.225,E2 -19727.225} C_VEL
LIN {X 0,Y 239.821,Z 583.416,A -85,B 0,C 180,E1 -19730.588,E2 -19730.588} C_VEL
LIN {X 0,Y 243.035,Z 574.869,A -85,B 0,C 180,E1 -19733.881,E2 -19733.881} C_VEL
LIN {X 0,Y 246.417,Z 565.772,A -85,B 0,C 180,E1 -19736.692,E2 -19736.692} C_VEL
LIN {X 0,Y 249.74,Z 556.352,A -85,B 0,C 180,E1 -19739.083,E2 -19739.083} C_VEL
LIN {X 0,Y 253.626,Z 544.496,A -85,B 0,C 180,E1 -19741.535,E2 -19741.535} C_VEL
LIN {X 0,Y 257.371,Z 532.221,A -85,B 0,C 180,E1 -19743.57,E2 -19743.57} C_VEL
LIN {X 0,Y 261.033,Z 518.667,A -85,B 0,C 180,E1 -19745.37,E2 -19745.37} C_VEL
LIN {X 0,Y 264.067,Z 504.738,A -85,B 0,C 180,E1 -19746.861,E2 -19746.861} C_VEL
LIN {X 0,Y 266.648,Z 490.596,A -85,B 0,C 180,E1 -19748.031,E2 -19748.031} C_VEL
LIN {X 0,Y 268.859,Z 475.074,A -85,B 0,C 180,E1 -19748.975,E2 -19748.975} C_VEL
LIN {X 0,Y 270.349,Z 459.614,A -85,B 0,C 180,E1 -19749.621,E2 -19749.621} C_VEL
LIN {X 0,Y 275.188,Z 367.164,A -85,B 0,C 180,E1 -19751.942,E2 -19751.942} C_VEL
LIN {X 0,Y 270.392,Z 357.086,A -85,B 0,C 180,E1 -19753.23,E2 -19753.23} C_VEL
LIN {X 0,Y 261.628,Z 342.149,A -85,B 0,C 180,E1 -19755.653,E2 -19755.653} C_VEL
LIN {X 0,Y 253.833,Z 330.341,A -85,B 0,C 180,E1 -19757.988,E2 -19757.988} C_VEL
LIN {X 0,Y 248.228,Z 322.402,A -85,B 0,C 180,E1 -19759.807,E2 -19759.807} C_VEL
LIN {X 0,Y 245.193,Z 318.305,A -85,B 0,C 180,E1 -19760.849,E2 -19760.849} C_VEL
LIN {X 0,Y 242.63,Z 314.728,A -85,B 0,C 180,E1 -19761.773,E2 -19761.773} C_VEL
LIN {X 0,Y 239.575,Z 311.018,A -85,B 0,C 180,E1 -19762.9,E2 -19762.9} C_VEL
LIN {X 0,Y 238.454,Z 309.096,A -85,B 0,C 180,E1 -19763.356,E2 -19763.356} C_VEL
LIN {X 0,Y 236.144,Z 306.986,A -85,B 0,C 180,E1 -19764.232,E2 -19764.232} C_VEL
LIN {X 0,Y 235.019,Z 304.444,A -85,B 0,C 180,E1 -19764.75,E2 -19764.75} C_VEL
LIN {X 0,Y 234.909,Z 303.816,A -85,B 0,C 180,E1 -19764.857,E2 -19764.857} C_VEL
LIN {X 0,Y 234.95,Z 303.842,A -85,B 0,C 180,E1 -19767.423,E2 -19767.423} C_VEL
LIN {X 0,Y 234.889,Z 303.847,A -85,B 0,C 180,E1 -19771.397,E2 -19771.397} C_VEL
LIN {X 0,Y 234.898,Z 303.848,A -85,B 0,C 180,E1 -19775.236,E2 -19775.236} C_VEL
LIN {X 0,Y 234.933,Z 303.847,A -85,B 0,C 180,E1 -19778.962,E2 -19778.962} C_VEL
LIN {X 0,Y 235.047,Z 303.831,A -85,B 0,C 180,E1 -19783.097,E2 -19783.097} C_VEL
LIN {X 0,Y 235.089,Z 303.825,A -85,B 0,C 180,E1 -19787.921,E2 -19787.921} C_VEL
LIN {X 0,Y 235.309,Z 303.784,A -85,B 0,C 180,E1 -19791.411,E2 -19791.411} C_VEL
LIN {X 0,Y 235.346,Z 303.795,A -85,B 0,C 180,E1 -19793.139,E2 -19793.139} C_VEL
LIN {X 0,Y 235.188,Z 303.801,A -85,B 0,C 180,E1 -19795.029,E2 -19795.029} C_VEL
LIN {X 0,Y 234.588,Z 303.875,A -85,B 0,C 180,E1 -19796.463,E2 -19796.463} C_VEL
LIN {X 0,Y 231.954,Z 304.217,A -85,B 0,C 180,E1 -19798.811,E2 -19798.811} C_VEL
LIN {X 0,Y 228.775,Z 304.599,A -85,B 0,C 180,E1 -19801.701,E2 -19801.701} C_VEL
LIN {X 0,Y 228.339,Z 304.657,A -85,B 0,C 180,E1 -19802.698,E2 -19802.698} C_VEL
LIN {X 0,Y 228.305,Z 304.66,A -85,B 0,C 180,E1 -19807.073,E2 -19807.073} C_VEL
LIN {X 0,Y 228.144,Z 304.677,A -85,B 0,C 180,E1 -19810.651,E2 -19810.651} C_VEL
LIN {X 0,Y 228.063,Z 304.693,A -85,B 0,C 180,E1 -19814.272,E2 -19814.272} C_VEL
LIN {X 0,Y 228.005,Z 304.708,A -85,B 0,C 180,E1 -19817.953,E2 -19817.953} C_VEL
LIN {X 0,Y 227.944,Z 304.708,A -85,B 0,C 180,E1 -19822.339,E2 -19822.339} C_VEL
LIN {X 0,Y 227.92,Z 304.683,A -85,B 0,C 180,E1 -19826.593,E2 -19826.593} C_VEL
LIN {X 0,Y 227.846,Z 304.76,A -85,B 0,C 180,E1 -19831.151,E2 -19831.151} C_VEL
LIN {X 0,Y 228.721,Z 307.181,A -85,B 0,C 180,E1 -19832.594,E2 -19832.594} C_VEL
LIN {X 0,Y 232.228,Z 312.134,A -85,B 0,C 180,E1 -19834.178,E2 -19834.178} C_VEL
LIN {X 0,Y 233.762,Z 314.292,A -85,B 0,C 180,E1 -19834.836,E2 -19834.836} C_VEL
LIN {X 0,Y 238.161,Z 320.652,A -85,B 0,C 180,E1 -19836.63,E2 -19836.63} C_VEL
LIN {X 0,Y 242.235,Z 327.018,A -85,B 0,C 180,E1 -19838.194,E2 -19838.194} C_VEL
LIN {X 0,Y 247.308,Z 335.038,A -85,B 0,C 180,E1 -19840.006,E2 -19840.006} C_VEL
LIN {X 0,Y 255.272,Z 349.208,A -85,B 0,C 180,E1 -19842.651,E2 -19842.651} C_VEL
LIN {X 0,Y 261.667,Z 362.08,A -85,B 0,C 180,E1 -19844.63,E2 -19844.63} C_VEL
LIN {X 0,Y 267.017,Z 374.124,A -85,B 0,C 180,E1 -19846.211,E2 -19846.211} C_VEL
LIN {X 0,Y 269.376,Z 379.966,A -85,B 0,C 180,E1 -19846.894,E2 -19846.894} C_VEL
LIN {X 0,Y 265.133,Z 460.856,A -85,B 0,C 180,E1 -19848.938,E2 -19848.938} C_VEL
LIN {X 0,Y 263.782,Z 480.197,A -85,B 0,C 180,E1 -19849.502,E2 -19849.502} C_VEL
LIN {X 0,Y 261.873,Z 495.568,A -85,B 0,C 180,E1 -19850.216,E2 -19850.216} C_VEL
LIN {X 0,Y 259.209,Z 510.413,A -85,B 0,C 180,E1 -19851.172,E2 -19851.172} C_VEL
LIN {X 0,Y 256.16,Z 524.337,A -85,B 0,C 180,E1 -19852.379,E2 -19852.379} C_VEL
LIN {X 0,Y 252.76,Z 537.685,A -85,B 0,C 180,E1 -19853.87,E2 -19853.87} C_VEL
LIN {X 0,Y 249.034,Z 550.363,A -85,B 0,C 180,E1 -19855.639,E2 -19855.639} C_VEL
LIN {X 0,Y 245.379,Z 561.426,A -85,B 0,C 180,E1 -19857.519,E2 -19857.519} C_VEL
LIN {X 0,Y 241.442,Z 572.615,A -85,B 0,C 180,E1 -19859.86,E2 -19859.86} C_VEL
LIN {X 0,Y 237.748,Z 582.739,A -85,B 0,C 180,E1 -19862.476,E2 -19862.476} C_VEL
LIN {X 0,Y 234.177,Z 592.55,A -85,B 0,C 180,E1 -19865.629,E2 -19865.629} C_VEL
LIN {X 0,Y 231.323,Z 600.076,A -85,B 0,C 180,E1 -19868.619,E2 -19868.619} C_VEL
LIN {X 0,Y 228.776,Z 607.328,A -85,B 0,C 180,E1 -19872.235,E2 -19872.235} C_VEL
LIN {X 0,Y 227.16,Z 612.649,A -85,B 0,C 180,E1 -19875.671,E2 -19875.671} C_VEL
LIN {X 0,Y 226.078,Z 616.845,A -85,B 0,C 180,E1 -19879.251,E2 -19879.251} C_VEL
LIN {X 0,Y 225.682,Z 619.8,A -85,B 0,C 180,E1 -19882.845,E2 -19882.845} C_VEL
LIN {X 0,Y 225.631,Z 621.566,A -85,B 0,C 180,E1 -19886.429,E2 -19886.429} C_VEL
LIN {X 0,Y 225.817,Z 622.176,A -85,B 0,C 180,E1 -19890.001,E2 -19890.001} C_VEL
LIN {X 0,Y 225.632,Z 621.552,A -85,B 0,C 180,E1 -19893.572,E2 -19893.572} C_VEL
LIN {X 0,Y 225.68,Z 619.768,A -85,B 0,C 180,E1 -19897.157,E2 -19897.157} C_VEL
LIN {X 0,Y 226.077,Z 616.8,A -85,B 0,C 180,E1 -19900.751,E2 -19900.751} C_VEL
LIN {X 0,Y 227.16,Z 612.592,A -85,B 0,C 180,E1 -19904.331,E2 -19904.331} C_VEL
LIN {X 0,Y 228.842,Z 607.029,A -85,B 0,C 180,E1 -19907.886,E2 -19907.886} C_VEL
LIN {X 0,Y 231.305,Z 599.968,A -85,B 0,C 180,E1 -19911.384,E2 -19911.384} C_VEL
LIN {X 0,Y 234.161,Z 592.431,A -85,B 0,C 180,E1 -19914.375,E2 -19914.375} C_VEL
LIN {X 0,Y 237.717,Z 582.653,A -85,B 0,C 180,E1 -19917.51,E2 -19917.51} C_VEL
LIN {X 0,Y 241.444,Z 572.444,A -85,B 0,C 180,E1 -19920.141,E2 -19920.141} C_VEL
LIN {X 0,Y 245.679,Z 560.195,A -85,B 0,C 180,E1 -19922.681,E2 -19922.681} C_VEL
LIN {X 0,Y 249.767,Z 547.717,A -85,B 0,C 180,E1 -19924.737,E2 -19924.737} C_VEL
LIN {X 0,Y 253.672,Z 533.808,A -85,B 0,C 180,E1 -19926.576,E2 -19926.576} C_VEL
LIN {X 0,Y 256.973,Z 520.344,A -85,B 0,C 180,E1 -19927.979,E2 -19927.979} C_VEL
LIN {X 0,Y 259.86,Z 506.541,A -85,B 0,C 180,E1 -19929.088,E2 -19929.088} C_VEL
LIN {X 0,Y 262.423,Z 491.081,A -85,B 0,C 180,E1 -19929.998,E2 -19929.998} C_VEL
LIN {X 0,Y 264.068,Z 475.766,A -85,B 0,C 180,E1 -19930.635,E2 -19930.635} C_VEL
LIN {X 0,Y 267.84,Z 407.429,A -85,B 0,C 180,E1 -19932.378,E2 -19932.378} C_VEL
LIN {X 0,Y 269.253,Z 379.842,A -85,B 0,C 180,E1 -19933.081,E2 -19933.081} C_VEL
LIN {X 0,Y 263.227,Z 365.452,A -85,B 0,C 180,E1 -19934.845,E2 -19934.845} C_VEL
LIN {X 0,Y 256.441,Z 351.531,A -85,B 0,C 180,E1 -19936.911,E2 -19936.911} C_VEL
LIN {X 0,Y 249.632,Z 339.106,A -85,B 0,C 180,E1 -19939.12,E2 -19939.12} C_VEL
LIN {X 0,Y 243.368,Z 328.731,A -85,B 0,C 180,E1 -19941.311,E2 -19941.311} C_VEL
LIN {X 0,Y 239.264,Z 322.455,A -85,B 0,C 180,E1 -19942.844,E2 -19942.844} C_VEL
LIN {X 0,Y 236.633,Z 318.39,A -85,B 0,C 180,E1 -19943.887,E2 -19943.887} C_VEL
LIN {X 0,Y 232.278,Z 312.187,A -85,B 0,C 180,E1 -19945.7,E2 -19945.7} C_VEL
LIN {X 0,Y 228.748,Z 307.285,A -85,B 0,C 180,E1 -19947.279,E2 -19947.279} C_VEL
LIN {X 0,Y 228.512,Z 306.81,A -85,B 0,C 180,E1 -19947.438,E2 -19947.438} C_VEL
LIN {X 0,Y 227.864,Z 304.721,A -85,B 0,C 180,E1 -19948.852,E2 -19948.852} C_VEL
LIN {X 0,Y 227.926,Z 304.706,A -85,B 0,C 180,E1 -19953.408,E2 -19953.408} C_VEL
LIN {X 0,Y 227.959,Z 304.707,A -85,B 0,C 180,E1 -19958.287,E2 -19958.287} C_VEL
LIN {X 0,Y 228.039,Z 304.705,A -85,B 0,C 180,E1 -19962.826,E2 -19962.826} C_VEL
LIN {X 0,Y 228.077,Z 304.695,A -85,B 0,C 180,E1 -19967.544,E2 -19967.544} C_VEL
LIN {X 0,Y 228.258,Z 304.678,A -85,B 0,C 180,E1 -19971.144,E2 -19971.144} C_VEL
LIN {X 0,Y 228.305,Z 304.659,A -85,B 0,C 180,E1 -19972.927,E2 -19972.927} C_VEL
LIN {X 0,Y 228.541,Z 304.633,A -85,B 0,C 180,E1 -19978.238,E2 -19978.238} C_VEL
LIN {X 0,Y 228.541,Z 304.63,A -85,B 0,C 180,E1 -19981.762,E2 -19981.762} C_VEL
LIN {X 0,Y 228.309,Z 304.662,A -85,B 0,C 180,E1 -19987.073,E2 -19987.073} C_VEL
LIN {X 0,Y 228.13,Z 304.681,A -85,B 0,C 180,E1 -19990.652,E2 -19990.652} C_VEL
LIN {X 0,Y 228.004,Z 304.704,A -85,B 0,C 180,E1 -19996.106,E2 -19996.106} C_VEL
LIN {X 0,Y 227.923,Z 304.713,A -85,B 0,C 180,E1 -20001.717,E2 -20001.717} C_VEL
LIN {X 0,Y 227.874,Z 304.697,A -85,B 0,C 180,E1 -20006.565,E2 -20006.565} C_VEL
LIN {X 0,Y 227.873,Z 304.708,A -85,B 0,C 180,E1 -20010.278,E2 -20010.278} C_VEL
LIN {X 0,Y 227.942,Z 304.887,A -85,B 0,C 180,E1 -20012.851,E2 -20012.851} C_VEL
LIN {X 0,Y 228.777,Z 307.378,A -85,B 0,C 180,E1 -20013.318,E2 -20013.318} C_VEL
LIN {X 0,Y 230.712,Z 309.566,A -85,B 0,C 180,E1 -20014.17,E2 -20014.17} C_VEL
LIN {X 0,Y 231.973,Z 310.499,A -85,B 0,C 180,E1 -20014.681,E2 -20014.681} C_VEL
LIN {X 0,Y 233.817,Z 313.576,A -85,B 0,C 180,E1 -20015.497,E2 -20015.497} C_VEL
LIN {X 0,Y 236.093,Z 315.964,A -85,B 0,C 180,E1 -20016.394,E2 -20016.394} C_VEL
LIN {X 0,Y 238.729,Z 319.556,A -85,B 0,C 180,E1 -20017.428,E2 -20017.428} C_VEL
LIN {X 0,Y 244.044,Z 326.845,A -85,B 0,C 180,E1 -20019.38,E2 -20019.38} C_VEL
LIN {X 0,Y 250.378,Z 335.886,A -85,B 0,C 180,E1 -20021.519,E2 -20021.519} C_VEL
LIN {X 0,Y 258.354,Z 348.293,A -85,B 0,C 180,E1 -20023.99,E2 -20023.99} C_VEL
LIN {X 0,Y 265.382,Z 360.478,A -85,B 0,C 180,E1 -20026.008,E2 -20026.008} C_VEL
LIN {X 0,Y 269.127,Z 368.084,A -85,B 0,C 180,E1 -20027.055,E2 -20027.055} C_VEL
LIN {X 0,Y 269.697,Z 369.468,A -85,B 0,C 180,E1 -20027.218,E2 -20027.218} C_VEL
LIN {X 0,Y 265.457,Z 449.917,A -85,B 0,C 180,E1 -20029.248,E2 -20029.248} C_VEL
LIN {X 0,Y 264.202,Z 466.511,A -85,B 0,C 180,E1 -20029.766,E2 -20029.766} C_VEL
LIN {X 0,Y 262.33,Z 482.054,A -85,B 0,C 180,E1 -20030.546,E2 -20030.546} C_VEL
LIN {X 0,Y 260.054,Z 496.334,A -85,B 0,C 180,E1 -20031.567,E2 -20031.567} C_VEL
LIN {X 0,Y 257.479,Z 509.19,A -85,B 0,C 180,E1 -20032.755,E2 -20032.755} C_VEL
LIN {X 0,Y 254.257,Z 522.409,A -85,B 0,C 180,E1 -20034.272,E2 -20034.272} C_VEL
LIN {X 0,Y 250.572,Z 535.33,A -85,B 0,C 180,E1 -20036.119,E2 -20036.119} C_VEL
LIN {X 0,Y 246.675,Z 547.128,A -85,B 0,C 180,E1 -20038.19,E2 -20038.19} C_VEL
LIN {X 0,Y 243.053,Z 557.907,A -85,B 0,C 180,E1 -20040.556,E2 -20040.556} C_VEL
LIN {X 0,Y 239.118,Z 568.391,A -85,B 0,C 180,E1 -20043.37,E2 -20043.37} C_VEL
LIN {X 0,Y 235.726,Z 577.098,A -85,B 0,C 180,E1 -20046.265,E2 -20046.265} C_VEL
LIN {X 0,Y 232.614,Z 584.901,A -85,B 0,C 180,E1 -20049.49,E2 -20049.49} C_VEL
LIN {X 0,Y 230.02,Z 591.768,A -85,B 0,C 180,E1 -20053.125,E2 -20053.125} C_VEL
LIN {X 0,Y 228.11,Z 596.863,A -85,B 0,C 180,E1 -20056.639,E2 -20056.639} C_VEL
LIN {X 0,Y 227.112,Z 599.794,A -85,B 0,C 180,E1 -20059.299,E2 -20059.299} C_VEL
LIN {X 0,Y 226.313,Z 602.655,A -85,B 0,C 180,E1 -20062.864,E2 -20062.864} C_VEL
LIN {X 0,Y 225.918,Z 604.372,A -85,B 0,C 180,E1 -20066.432,E2 -20066.432} C_VEL
LIN {X 0,Y 225.832,Z 604.969,A -85,B 0,C 180,E1 -20069.999,E2 -20069.999} C_VEL
LIN {X 0,Y 225.918,Z 604.41,A -85,B 0,C 180,E1 -20073.566,E2 -20073.566} C_VEL
LIN {X 0,Y 226.312,Z 602.743,A -85,B 0,C 180,E1 -20077.135,E2 -20077.135} C_VEL
LIN {X 0,Y 227.101,Z 599.928,A -85,B 0,C 180,E1 -20080.7,E2 -20080.7} C_VEL
LIN {X 0,Y 228.441,Z 595.891,A -85,B 0,C 180,E1 -20084.247,E2 -20084.247} C_VEL
LIN {X 0,Y 230.52,Z 590.526,A -85,B 0,C 180,E1 -20087.75,E2 -20087.75} C_VEL
LIN {X 0,Y 233.159,Z 583.686,A -85,B 0,C 180,E1 -20091.204,E2 -20091.204} C_VEL
LIN {X 0,Y 236.527,Z 575.138,A -85,B 0,C 180,E1 -20094.581,E2 -20094.581} C_VEL
LIN {X 0,Y 240.089,Z 566.04,A -85,B 0,C 180,E1 -20097.454,E2 -20097.454} C_VEL
LIN {X 0,Y 243.376,Z 557.041,A -85,B 0,C 180,E1 -20099.796,E2 -20099.796} C_VEL
LIN {X 0,Y 247.238,Z 545.752,A -85,B 0,C 180,E1 -20102.207,E2 -20102.207} C_VEL
LIN {X 0,Y 251.147,Z 533.669,A -85,B 0,C 180,E1 -20104.275,E2 -20104.275} C_VEL
LIN {X 0,Y 254.903,Z 520.396,A -85,B 0,C 180,E1 -20106.109,E2 -20106.109} C_VEL
LIN {X 0,Y 257.952,Z 507.233,A -85,B 0,C 180,E1 -20107.581,E2 -20107.581} C_VEL
LIN {X 0,Y 260.748,Z 493.129,A -85,B 0,C 180,E1 -20108.804,E2 -20108.804} C_VEL
LIN {X 0,Y 262.931,Z 478.468,A -85,B 0,C 180,E1 -20109.779,E2 -20109.779} C_VEL
LIN {X 0,Y 264.647,Z 463.426,A -85,B 0,C 180,E1 -20110.463,E2 -20110.463} C_VEL
LIN {X 0,Y 265.88,Z 445.09,A -85,B 0,C 180,E1 -20110.985,E2 -20110.985} C_VEL
LIN {X 0,Y 269.842,Z 370.399,A -85,B 0,C 180,E1 -20112.864,E2 -20112.864} C_VEL
LIN {X 0,Y 269.581,Z 368.871,A -85,B 0,C 180,E1 -20112.971,E2 -20112.971} C_VEL
LIN {X 0,Y 265.329,Z 360.227,A -85,B 0,C 180,E1 -20114.159,E2 -20114.159} C_VEL
LIN {X 0,Y 257.271,Z 346.447,A -85,B 0,C 180,E1 -20116.492,E2 -20116.492} C_VEL
LIN {X 0,Y 250.22,Z 335.584,A -85,B 0,C 180,E1 -20118.698,E2 -20118.698} C_VEL
LIN {X 0,Y 244.725,Z 327.733,A -85,B 0,C 180,E1 -20120.554,E2 -20120.554} C_VEL
LIN {X 0,Y 241.765,Z 323.703,A -85,B 0,C 180,E1 -20121.611,E2 -20121.611} C_VEL
LIN {X 0,Y 238.69,Z 319.522,A -85,B 0,C 180,E1 -20122.766,E2 -20122.766} C_VEL
LIN {X 0,Y 236.005,Z 315.825,A -85,B 0,C 180,E1 -20123.827,E2 -20123.827} C_VEL
LIN {X 0,Y 232.796,Z 312.097,A -85,B 0,C 180,E1 -20125.13,E2 -20125.13} C_VEL
LIN {X 0,Y 231.748,Z 310.191,A -85,B 0,C 180,E1 -20125.61,E2 -20125.61} C_VEL
LIN {X 0,Y 229.391,Z 308.279,A -85,B 0,C 180,E1 -20126.595,E2 -20126.595} C_VEL
LIN {X 0,Y 228.101,Z 305.734,A -85,B 0,C 180,E1 -20127.24,E2 -20127.24} C_VEL
LIN {X 0,Y 227.91,Z 304.718,A -85,B 0,C 180,E1 -20127.471,E2 -20127.471} C_VEL
LIN {X 0,Y 227.869,Z 304.726,A -85,B 0,C 180,E1 -20130.43,E2 -20130.43} C_VEL
LIN {X 0,Y 227.864,Z 304.727,A -85,B 0,C 180,E1 -20134.418,E2 -20134.418} C_VEL
LIN {X 0,Y 227.917,Z 304.717,A -85,B 0,C 180,E1 -20138.282,E2 -20138.282} C_VEL
LIN {X 0,Y 228.007,Z 304.709,A -85,B 0,C 180,E1 -20143.894,E2 -20143.894} C_VEL
LIN {X 0,Y 228.138,Z 304.686,A -85,B 0,C 180,E1 -20149.348,E2 -20149.348} C_VEL
LIN {X 0,Y 228.299,Z 304.671,A -85,B 0,C 180,E1 -20152.927,E2 -20152.927} C_VEL
LIN {X 0,Y 228.537,Z 304.643,A -85,B 0,C 180,E1 -20158.238,E2 -20158.238} C_VEL
LIN {X 0,Y 228.537,Z 304.627,A -85,B 0,C 180,E1 -20161.762,E2 -20161.762} C_VEL
LIN {X 0,Y 228.339,Z 304.657,A -85,B 0,C 180,E1 -20162.698,E2 -20162.698} C_VEL
LIN {X 0,Y 227.509,Z 304.772,A -85,B 0,C 180,E1 -20164.169,E2 -20164.169} C_VEL
LIN {X 0,Y 224.642,Z 305.127,A -85,B 0,C 180,E1 -20166.573,E2 -20166.573} C_VEL
LIN {X 0,Y 221.461,Z 305.516,A -85,B 0,C 180,E1 -20169.539,E2 -20169.539} C_VEL
LIN {X 0,Y 221.096,Z 305.554,A -85,B 0,C 180,E1 -20170.566,E2 -20170.566} C_VEL
LIN {X 0,Y 220.994,Z 305.57,A -85,B 0,C 180,E1 -20174.739,E2 -20174.739} C_VEL
LIN {X 0,Y 220.925,Z 305.584,A -85,B 0,C 180,E1 -20178.549,E2 -20178.549} C_VEL
LIN {X 0,Y 220.887,Z 305.578,A -85,B 0,C 180,E1 -20182.678,E2 -20182.678} C_VEL
LIN {X 0,Y 220.863,Z 305.566,A -85,B 0,C 180,E1 -20187.005,E2 -20187.005} C_VEL
LIN {X 0,Y 220.822,Z 305.801,A -85,B 0,C 180,E1 -20188.905,E2 -20188.905} C_VEL
LIN {X 0,Y 221.039,Z 306.615,A -85,B 0,C 180,E1 -20189.33,E2 -20189.33} C_VEL
LIN {X 0,Y 222.307,Z 309.116,A -85,B 0,C 180,E1 -20190.058,E2 -20190.058} C_VEL
LIN {X 0,Y 225.886,Z 312.923,A -85,B 0,C 180,E1 -20191.801,E2 -20191.801} C_VEL
LIN {X 0,Y 229.635,Z 318.234,A -85,B 0,C 180,E1 -20193.559,E2 -20193.559} C_VEL
LIN {X 0,Y 235.118,Z 326.378,A -85,B 0,C 180,E1 -20195.921,E2 -20195.921} C_VEL
LIN {X 0,Y 241.595,Z 336.667,A -85,B 0,C 180,E1 -20198.454,E2 -20198.454} C_VEL
LIN {X 0,Y 249.051,Z 349.722,A -85,B 0,C 180,E1 -20201.109,E2 -20201.109} C_VEL
LIN {X 0,Y 255.766,Z 362.966,A -85,B 0,C 180,E1 -20203.321,E2 -20203.321} C_VEL
LIN {X 0,Y 261.798,Z 376.401,A -85,B 0,C 180,E1 -20205.201,E2 -20205.201} C_VEL
LIN {X 0,Y 264.051,Z 382.123,A -85,B 0,C 180,E1 -20205.892,E2 -20205.892} C_VEL
LIN {X 0,Y 260.411,Z 449.861,A -85,B 0,C 180,E1 -20207.635,E2 -20207.635} C_VEL
LIN {X 0,Y 258.75,Z 476.516,A -85,B 0,C 180,E1 -20208.349,E2 -20208.349} C_VEL
LIN {X 0,Y 257.045,Z 491.491,A -85,B 0,C 180,E1 -20208.99,E2 -20208.99} C_VEL
LIN {X 0,Y 254.408,Z 506.753,A -85,B 0,C 180,E1 -20209.91,E2 -20209.91} C_VEL
LIN {X 0,Y 251.429,Z 520.501,A -85,B 0,C 180,E1 -20211.03,E2 -20211.03} C_VEL
LIN {X 0,Y 248.024,Z 533.792,A -85,B 0,C 180,E1 -20212.438,E2 -20212.438} C_VEL
LIN {X 0,Y 244.369,Z 546.413,A -85,B 0,C 180,E1 -20214.129,E2 -20214.129} C_VEL
LIN {X 0,Y 240.107,Z 559.068,A -85,B 0,C 180,E1 -20216.212,E2 -20216.212} C_VEL
LIN {X 0,Y 235.935,Z 570.578,A -85,B 0,C 180,E1 -20218.582,E2 -20218.582} C_VEL
LIN {X 0,Y 232.25,Z 580.275,A -85,B 0,C 180,E1 -20221.043,E2 -20221.043} C_VEL
LIN {X 0,Y 228.607,Z 589.814,A -85,B 0,C 180,E1 -20224.019,E2 -20224.019} C_VEL
LIN {X 0,Y 225.417,Z 597.765,A -85,B 0,C 180,E1 -20227.064,E2 -20227.064} C_VEL
LIN {X 0,Y 222.563,Z 605.2,A -85,B 0,C 180,E1 -20230.637,E2 -20230.637} C_VEL
LIN {X 0,Y 220.571,Z 611.112,A -85,B 0,C 180,E1 -20234.287,E2 -20234.287} C_VEL
LIN {X 0,Y 219.522,Z 614.634,A -85,B 0,C 180,E1 -20237.051,E2 -20237.051} C_VEL
LIN {X 0,Y 218.74,Z 618.202,A -85,B 0,C 180,E1 -20240.756,E2 -20240.756} C_VEL
LIN {X 0,Y 218.56,Z 620.559,A -85,B 0,C 180,E1 -20244.465,E2 -20244.465} C_VEL
LIN {X 0,Y 218.621,Z 621.747,A -85,B 0,C 180,E1 -20248.159,E2 -20248.159} C_VEL
LIN {X 0,Y 218.727,Z 621.906,A -85,B 0,C 180,E1 -20250.001,E2 -20250.001} C_VEL
LIN {X 0,Y 218.531,Z 621.281,A -85,B 0,C 180,E1 -20253.689,E2 -20253.689} C_VEL
LIN {X 0,Y 218.595,Z 619.495,A -85,B 0,C 180,E1 -20257.39,E2 -20257.39} C_VEL
LIN {X 0,Y 219.061,Z 616.527,A -85,B 0,C 180,E1 -20261.099,E2 -20261.099} C_VEL
LIN {X 0,Y 220.225,Z 612.318,A -85,B 0,C 180,E1 -20264.792,E2 -20264.792} C_VEL
LIN {X 0,Y 222.01,Z 606.754,A -85,B 0,C 180,E1 -20268.456,E2 -20268.456} C_VEL
LIN {X 0,Y 224.604,Z 599.692,A -85,B 0,C 180,E1 -20272.055,E2 -20272.055} C_VEL
LIN {X 0,Y 227.651,Z 592.156,A -85,B 0,C 180,E1 -20275.119,E2 -20275.119} C_VEL
LIN {X 0,Y 231.11,Z 583.052,A -85,B 0,C 180,E1 -20278.13,E2 -20278.13} C_VEL
LIN {X 0,Y 235.286,Z 572.169,A -85,B 0,C 180,E1 -20281.016,E2 -20281.016} C_VEL
LIN {X 0,Y 239.71,Z 559.92,A -85,B 0,C 180,E1 -20283.601,E2 -20283.601} C_VEL
LIN {X 0,Y 243.956,Z 547.442,A -85,B 0,C 180,E1 -20285.689,E2 -20285.689} C_VEL
LIN {X 0,Y 247.791,Z 534.255,A -85,B 0,C 180,E1 -20287.475,E2 -20287.475} C_VEL
LIN {X 0,Y 251.393,Z 520.066,A -85,B 0,C 180,E1 -20288.979,E2 -20288.979} C_VEL
LIN {X 0,Y 254.396,Z 506.263,A -85,B 0,C 180,E1 -20290.095,E2 -20290.095} C_VEL
LIN {X 0,Y 257.033,Z 490.801,A -85,B 0,C 180,E1 -20291.014,E2 -20291.014} C_VEL
LIN {X 0,Y 258.713,Z 475.479,A -85,B 0,C 180,E1 -20291.66,E2 -20291.66} C_VEL
LIN {X 0,Y 262.474,Z 409.896,A -85,B 0,C 180,E1 -20293.354,E2 -20293.354} C_VEL
LIN {X 0,Y 263.903,Z 381.891,A -85,B 0,C 180,E1 -20294.09,E2 -20294.09} C_VEL
LIN {X 0,Y 258.334,Z 368.548,A -85,B 0,C 180,E1 -20295.803,E2 -20295.803} C_VEL
LIN {X 0,Y 252.082,Z 355.601,A -85,B 0,C 180,E1 -20297.801,E2 -20297.801} C_VEL
LIN {X 0,Y 245.881,Z 344.102,A -85,B 0,C 180,E1 -20299.909,E2 -20299.909} C_VEL
LIN {X 0,Y 239.772,Z 333.821,A -85,B 0,C 180,E1 -20302.143,E2 -20302.143} C_VEL
LIN {X 0,Y 233.704,Z 324.229,A -85,B 0,C 180,E1 -20304.57,E2 -20304.57} C_VEL
LIN {X 0,Y 229.345,Z 317.944,A -85,B 0,C 180,E1 -20306.458,E2 -20306.458} C_VEL
LIN {X 0,Y 225.075,Z 312.028,A -85,B 0,C 180,E1 -20308.465,E2 -20308.465} C_VEL
LIN {X 0,Y 221.645,Z 308.117,A -85,B 0,C 180,E1 -20310.17,E2 -20310.17} C_VEL
LIN {X 0,Y 220.962,Z 306.359,A -85,B 0,C 180,E1 -20310.593,E2 -20310.593} C_VEL
LIN {X 0,Y 220.808,Z 305.593,A -85,B 0,C 180,E1 -20311.223,E2 -20311.223} C_VEL
LIN {X 0,Y 220.879,Z 305.583,A -85,B 0,C 180,E1 -20313.548,E2 -20313.548} C_VEL
LIN {X 0,Y 220.872,Z 305.585,A -85,B 0,C 180,E1 -20317.553,E2 -20317.553} C_VEL
LIN {X 0,Y 220.989,Z 305.583,A -85,B 0,C 180,E1 -20322.572,E2 -20322.572} C_VEL
LIN {X 0,Y 221.016,Z 305.579,A -85,B 0,C 180,E1 -20327.139,E2 -20327.139} C_VEL
LIN {X 0,Y 221.199,Z 305.557,A -85,B 0,C 180,E1 -20330.859,E2 -20330.859} C_VEL
LIN {X 0,Y 221.243,Z 305.539,A -85,B 0,C 180,E1 -20332.7,E2 -20332.7} C_VEL
LIN {X 0,Y 221.474,Z 305.513,A -85,B 0,C 180,E1 -20338.182,E2 -20338.182} C_VEL
LIN {X 0,Y 221.475,Z 305.51,A -85,B 0,C 180,E1 -20341.819,E2 -20341.819} C_VEL
LIN {X 0,Y 221.247,Z 305.544,A -85,B 0,C 180,E1 -20347.3,E2 -20347.3} C_VEL
LIN {X 0,Y 221.055,Z 305.563,A -85,B 0,C 180,E1 -20350.997,E2 -20350.997} C_VEL
LIN {X 0,Y 220.97,Z 305.586,A -85,B 0,C 180,E1 -20356.634,E2 -20356.634} C_VEL
LIN {X 0,Y 220.85,Z 305.6,A -85,B 0,C 180,E1 -20360.49,E2 -20360.49} C_VEL
LIN {X 0,Y 220.825,Z 305.604,A -85,B 0,C 180,E1 -20364.44,E2 -20364.44} C_VEL
LIN {X 0,Y 220.795,Z 305.569,A -85,B 0,C 180,E1 -20368.52,E2 -20368.52} C_VEL
LIN {X 0,Y 220.834,Z 305.615,A -85,B 0,C 180,E1 -20369.885,E2 -20369.885} C_VEL
LIN {X 0,Y 221.751,Z 308.321,A -85,B 0,C 180,E1 -20370.471,E2 -20370.471} C_VEL
LIN {X 0,Y 223.76,Z 310.526,A -85,B 0,C 180,E1 -20371.478,E2 -20371.478} C_VEL
LIN {X 0,Y 225.146,Z 311.409,A -85,B 0,C 180,E1 -20372.108,E2 -20372.108} C_VEL
LIN {X 0,Y 226.901,Z 314.487,A -85,B 0,C 180,E1 -20372.993,E2 -20372.993} C_VEL
LIN {X 0,Y 229.338,Z 316.94,A -85,B 0,C 180,E1 -20374.065,E2 -20374.065} C_VEL
LIN {X 0,Y 231.846,Z 320.442,A -85,B 0,C 180,E1 -20375.167,E2 -20375.167} C_VEL
LIN {X 0,Y 233.289,Z 322.098,A -85,B 0,C 180,E1 -20375.758,E2 -20375.758} C_VEL
LIN {X 0,Y 237.442,Z 327.83,A -85,B 0,C 180,E1 -20377.424,E2 -20377.424} C_VEL
LIN {X 0,Y 243.074,Z 335.611,A -85,B 0,C 180,E1 -20379.501,E2 -20379.501} C_VEL
LIN {X 0,Y 250.686,Z 347.154,A -85,B 0,C 180,E1 -20382.076,E2 -20382.076} C_VEL
LIN {X 0,Y 257.989,Z 359.346,A -85,B 0,C 180,E1 -20384.34,E2 -20384.34} C_VEL
LIN {X 0,Y 263.442,Z 369.631,A -85,B 0,C 180,E1 -20385.938,E2 -20385.938} C_VEL
LIN {X 0,Y 264.428,Z 371.781,A -85,B 0,C 180,E1 -20386.226,E2 -20386.226} C_VEL
LIN {X 0,Y 259.529,Z 459.706,A -85,B 0,C 180,E1 -20388.5,E2 -20388.5} C_VEL
LIN {X 0,Y 257.861,Z 475.358,A -85,B 0,C 180,E1 -20389.146,E2 -20389.146} C_VEL
LIN {X 0,Y 255.769,Z 489.665,A -85,B 0,C 180,E1 -20390.036,E2 -20390.036} C_VEL
LIN {X 0,Y 252.927,Z 504.359,A -85,B 0,C 180,E1 -20391.251,E2 -20391.251} C_VEL
LIN {X 0,Y 249.718,Z 518.289,A -85,B 0,C 180,E1 -20392.764,E2 -20392.764} C_VEL
LIN {X 0,Y 245.799,Z 532.03,A -85,B 0,C 180,E1 -20394.619,E2 -20394.619} C_VEL
LIN {X 0,Y 241.73,Z 544.425,A -85,B 0,C 180,E1 -20396.717,E2 -20396.717} C_VEL
LIN {X 0,Y 238.023,Z 554.844,A -85,B 0,C 180,E1 -20398.901,E2 -20398.901} C_VEL
LIN {X 0,Y 234.467,Z 564.407,A -85,B 0,C 180,E1 -20401.34,E2 -20401.34} C_VEL
LIN {X 0,Y 230.668,Z 573.827,A -85,B 0,C 180,E1 -20404.266,E2 -20404.266} C_VEL
LIN {X 0,Y 227.392,Z 581.664,A -85,B 0,C 180,E1 -20407.272,E2 -20407.272} C_VEL
LIN {X 0,Y 224.417,Z 588.969,A -85,B 0,C 180,E1 -20410.802,E2 -20410.802} C_VEL
LIN {X 0,Y 222.039,Z 594.761,A -85,B 0,C 180,E1 -20414.392,E2 -20414.392} C_VEL
LIN {X 0,Y 220.805,Z 598.182,A -85,B 0,C 180,E1 -20417.125,E2 -20417.125} C_VEL
LIN {X 0,Y 219.594,Z 601.644,A -85,B 0,C 180,E1 -20420.791,E2 -20420.791} C_VEL
LIN {X 0,Y 218.995,Z 603.925,A -85,B 0,C 180,E1 -20424.474,E2 -20424.474} C_VEL
LIN {X 0,Y 218.762,Z 605.085,A -85,B 0,C 180,E1 -20428.158,E2 -20428.158} C_VEL
LIN {X 0,Y 218.761,Z 605.097,A -85,B 0,C 180,E1 -20431.84,E2 -20431.84} C_VEL
LIN {X 0,Y 219.044,Z 603.812,A -85,B 0,C 180,E1 -20435.938,E2 -20435.938} C_VEL
LIN {X 0,Y 219.591,Z 601.755,A -85,B 0,C 180,E1 -20439.207,E2 -20439.207} C_VEL
LIN {X 0,Y 220.77,Z 598.337,A -85,B 0,C 180,E1 -20442.875,E2 -20442.875} C_VEL
LIN {X 0,Y 222.538,Z 593.653,A -85,B 0,C 180,E1 -20446.512,E2 -20446.512} C_VEL
LIN {X 0,Y 224.984,Z 587.576,A -85,B 0,C 180,E1 -20450.096,E2 -20450.096} C_VEL
LIN {X 0,Y 228.201,Z 579.913,A -85,B 0,C 180,E1 -20453.6,E2 -20453.6} C_VEL
LIN {X 0,Y 231.621,Z 571.735,A -85,B 0,C 180,E1 -20456.586,E2 -20456.586} C_VEL
LIN {X 0,Y 235.613,Z 561.874,A -85,B 0,C 180,E1 -20459.483,E2 -20459.483} C_VEL
LIN {X 0,Y 238.85,Z 552.873,A -85,B 0,C 180,E1 -20461.671,E2 -20461.671} C_VEL
LIN {X 0,Y 242.749,Z 541.841,A -85,B 0,C 180,E1 -20463.87,E2 -20463.87} C_VEL
LIN {X 0,Y 246.787,Z 528.909,A -85,B 0,C 180,E1 -20465.969,E2 -20465.969} C_VEL
LIN {X 0,Y 250.344,Z 516.05,A -85,B 0,C 180,E1 -20467.632,E2 -20467.632} C_VEL
LIN {X 0,Y 253.469,Z 502.224,A -85,B 0,C 180,E1 -20469.071,E2 -20469.071} C_VEL
LIN {X 0,Y 256.276,Z 487.243,A -85,B 0,C 180,E1 -20470.252,E2 -20470.252} C_VEL
LIN {X 0,Y 258.328,Z 472.85,A -85,B 0,C 180,E1 -20471.085,E2 -20471.085} C_VEL
LIN {X 0,Y 259.685,Z 458.612,A -85,B 0,C 180,E1 -20471.662,E2 -20471.662} C_VEL
LIN {X 0,Y 264.518,Z 373.346,A -85,B 0,C 180,E1 -20473.844,E2 -20473.844} C_VEL
LIN {X 0,Y 264.406,Z 371.541,A -85,B 0,C 180,E1 -20473.934,E2 -20473.934} C_VEL
LIN {X 0,Y 260.21,Z 363.147,A -85,B 0,C 180,E1 -20475.162,E2 -20475.162} C_VEL
LIN {X 0,Y 252.808,Z 350.499,A -85,B 0,C 180,E1 -20477.41,E2 -20477.41} C_VEL
LIN {X 0,Y 244.905,Z 338.169,A -85,B 0,C 180,E1 -20480.031,E2 -20480.031} C_VEL
LIN {X 0,Y 238.562,Z 329.298,A -85,B 0,C 180,E1 -20482.329,E2 -20482.329} C_VEL
LIN {X 0,Y 235.388,Z 324.99,A -85,B 0,C 180,E1 -20483.569,E2 -20483.569} C_VEL
LIN {X 0,Y 232.329,Z 320.85,A -85,B 0,C 180,E1 -20484.831,E2 -20484.831} C_VEL
LIN {X 0,Y 229.661,Z 317.456,A -85,B 0,C 180,E1 -20485.983,E2 -20485.983} C_VEL
LIN {X 0,Y 228.923,Z 316.349,A -85,B 0,C 180,E1 -20486.322,E2 -20486.322} C_VEL
LIN {X 0,Y 226.39,Z 313.792,A -85,B 0,C 180,E1 -20487.454,E2 -20487.454} C_VEL
LIN {X 0,Y 224.972,Z 311.176,A -85,B 0,C 180,E1 -20488.186,E2 -20488.186} C_VEL
LIN {X 0,Y 222.552,Z 309.445,A -85,B 0,C 180,E1 -20489.323,E2 -20489.323} C_VEL
LIN {X 0,Y 221.157,Z 307.049,A -85,B 0,C 180,E1 -20490.097,E2 -20490.097} C_VEL
LIN {X 0,Y 220.841,Z 305.601,A -85,B 0,C 180,E1 -20490.379,E2 -20490.379} C_VEL
LIN {X 0,Y 220.826,Z 305.595,A -85,B 0,C 180,E1 -20493.54,E2 -20493.54} C_VEL
LIN {X 0,Y 220.852,Z 305.589,A -85,B 0,C 180,E1 -20497.55,E2 -20497.55} C_VEL
LIN {X 0,Y 220.913,Z 305.585,A -85,B 0,C 180,E1 -20502.629,E2 -20502.629} C_VEL
LIN {X 0,Y 220.977,Z 305.574,A -85,B 0,C 180,E1 -20507.136,E2 -20507.136} C_VEL
LIN {X 0,Y 221.192,Z 305.54,A -85,B 0,C 180,E1 -20510.859,E2 -20510.859} C_VEL
LIN {X 0,Y 221.113,Z 305.559,A -85,B 0,C 180,E1 -20514.528,E2 -20514.528} C_VEL
LIN {X 0,Y 221.47,Z 305.522,A -85,B 0,C 180,E1 -20518.181,E2 -20518.181} C_VEL
LIN {X 0,Y 221.47,Z 305.507,A -85,B 0,C 180,E1 -20521.818,E2 -20521.818} C_VEL
LIN {X 0,Y 221.242,Z 305.542,A -85,B 0,C 180,E1 -20527.3,E2 -20527.3} C_VEL
LIN {X 0,Y 221.096,Z 305.554,A -85,B 0,C 180,E1 -20530.566,E2 -20530.566} C_VEL
LIN {X 0,Y 220.339,Z 305.659,A -85,B 0,C 180,E1 -20532.085,E2 -20532.085} C_VEL
LIN {X 0,Y 217.438,Z 306.02,A -85,B 0,C 180,E1 -20534.563,E2 -20534.563} C_VEL
LIN {X 0,Y 215.013,Z 306.325,A -85,B 0,C 180,E1 -20536.587,E2 -20536.587} C_VEL
LIN {X 0,Y 213.968,Z 306.455,A -85,B 0,C 180,E1 -20538.159,E2 -20538.159} C_VEL
LIN {X 0,Y 213.876,Z 306.46,A -85,B 0,C 180,E1 -20538.692,E2 -20538.692} C_VEL
LIN {X 0,Y 213.809,Z 306.448,A -85,B 0,C 180,E1 -20543.231,E2 -20543.231} C_VEL
LIN {X 0,Y 213.791,Z 306.457,A -85,B 0,C 180,E1 -20545.691,E2 -20545.691} C_VEL
LIN {X 0,Y 214.591,Z 308.886,A -85,B 0,C 180,E1 -20546.305,E2 -20546.305} C_VEL
LIN {X 0,Y 216.635,Z 311.285,A -85,B 0,C 180,E1 -20547.535,E2 -20547.535} C_VEL
LIN {X 0,Y 218.371,Z 312.529,A -85,B 0,C 180,E1 -20548.471,E2 -20548.471} C_VEL
LIN {X 0,Y 220.268,Z 315.682,A -85,B 0,C 180,E1 -20549.563,E2 -20549.563} C_VEL
LIN {X 0,Y 223.588,Z 319.413,A -85,B 0,C 180,E1 -20551.241,E2 -20551.241} C_VEL
LIN {X 0,Y 228.368,Z 326.484,A -85,B 0,C 180,E1 -20553.541,E2 -20553.541} C_VEL
LIN {X 0,Y 232.1,Z 332.097,A -85,B 0,C 180,E1 -20555.189,E2 -20555.189} C_VEL
LIN {X 0,Y 238.436,Z 342.418,A -85,B 0,C 180,E1 -20557.773,E2 -20557.773} C_VEL
LIN {X 0,Y 245.688,Z 355.507,A -85,B 0,C 180,E1 -20560.465,E2 -20560.465} C_VEL
LIN {X 0,Y 252.204,Z 368.657,A -85,B 0,C 180,E1 -20562.697,E2 -20562.697} C_VEL
LIN {X 0,Y 257.915,Z 381.961,A -85,B 0,C 180,E1 -20564.561,E2 -20564.561} C_VEL
LIN {X 0,Y 258.926,Z 384.598,A -85,B 0,C 180,E1 -20564.887,E2 -20564.887} C_VEL
LIN {X 0,Y 253.631,Z 475.06,A -85,B 0,C 180,E1 -20567.244,E2 -20567.244} C_VEL
LIN {X 0,Y 251.707,Z 491.229,A -85,B 0,C 180,E1 -20567.925,E2 -20567.925} C_VEL
LIN {X 0,Y 249.016,Z 506.489,A -85,B 0,C 180,E1 -20568.857,E2 -20568.857} C_VEL
LIN {X 0,Y 245.931,Z 520.235,A -85,B 0,C 180,E1 -20569.986,E2 -20569.986} C_VEL
LIN {X 0,Y 242.254,Z 534.113,A -85,B 0,C 180,E1 -20571.479,E2 -20571.479} C_VEL
LIN {X 0,Y 238.218,Z 547.44,A -85,B 0,C 180,E1 -20573.315,E2 -20573.315} C_VEL
LIN {X 0,Y 233.828,Z 559.874,A -85,B 0,C 180,E1 -20575.438,E2 -20575.438} C_VEL
LIN {X 0,Y 229.187,Z 572.076,A -85,B 0,C 180,E1 -20578.065,E2 -20578.065} C_VEL
LIN {X 0,Y 225.082,Z 582.373,A -85,B 0,C 180,E1 -20580.845,E2 -20580.845} C_VEL
LIN {X 0,Y 221.166,Z 592.006,A -85,B 0,C 180,E1 -20584.092,E2 -20584.092} C_VEL
LIN {X 0,Y 217.987,Z 599.53,A -85,B 0,C 180,E1 -20587.24,E2 -20587.24} C_VEL
LIN {X 0,Y 215.198,Z 606.562,A -85,B 0,C 180,E1 -20590.939,E2 -20590.939} C_VEL
LIN {X 0,Y 213.271,Z 612.103,A -85,B 0,C 180,E1 -20594.715,E2 -20594.715} C_VEL
LIN {X 0,Y 212.044,Z 616.302,A -85,B 0,C 180,E1 -20598.53,E2 -20598.53} C_VEL
LIN {X 0,Y 211.514,Z 619.256,A -85,B 0,C 180,E1 -20602.363,E2 -20602.363} C_VEL
LIN {X 0,Y 211.435,Z 621.025,A -85,B 0,C 180,E1 -20606.189,E2 -20606.189} C_VEL
LIN {X 0,Y 211.639,Z 621.636,A -85,B 0,C 180,E1 -20610.001,E2 -20610.001} C_VEL
LIN {X 0,Y 211.436,Z 621.01,A -85,B 0,C 180,E1 -20613.813,E2 -20613.813} C_VEL
LIN {X 0,Y 211.513,Z 619.223,A -85,B 0,C 180,E1 -20617.639,E2 -20617.639} C_VEL
LIN {X 0,Y 212.042,Z 616.254,A -85,B 0,C 180,E1 -20621.472,E2 -20621.472} C_VEL
LIN {X 0,Y 213.271,Z 612.043,A -85,B 0,C 180,E1 -20625.286,E2 -20625.286} C_VEL
LIN {X 0,Y 215.2,Z 606.479,A -85,B 0,C 180,E1 -20629.062,E2 -20629.062} C_VEL
LIN {X 0,Y 217.96,Z 599.417,A -85,B 0,C 180,E1 -20632.765,E2 -20632.765} C_VEL
LIN {X 0,Y 221.162,Z 591.88,A -85,B 0,C 180,E1 -20635.91,E2 -20635.91} C_VEL
LIN {X 0,Y 224.952,Z 582.478,A -85,B 0,C 180,E1 -20639.083,E2 -20639.083} C_VEL
LIN {X 0,Y 229.192,Z 571.895,A -85,B 0,C 180,E1 -20641.936,E2 -20641.936} C_VEL
LIN {X 0,Y 233.799,Z 559.645,A -85,B 0,C 180,E1 -20644.569,E2 -20644.569} C_VEL
LIN {X 0,Y 238.214,Z 547.167,A -85,B 0,C 180,E1 -20646.687,E2 -20646.687} C_VEL
LIN {X 0,Y 241.949,Z 534.734,A -85,B 0,C 180,E1 -20648.411,E2 -20648.411} C_VEL
LIN {X 0,Y 245.911,Z 519.79,A -85,B 0,C 180,E1 -20650.02,E2 -20650.02} C_VEL
LIN {X 0,Y 248.987,Z 505.985,A -85,B 0,C 180,E1 -20651.151,E2 -20651.151} C_VEL
LIN {X 0,Y 251.702,Z 490.519,A -85,B 0,C 180,E1 -20652.078,E2 -20652.078} C_VEL
LIN {X 0,Y 253.444,Z 475.193,A -85,B 0,C 180,E1 -20652.729,E2 -20652.729} C_VEL
LIN {X 0,Y 257.282,Z 411.068,A -85,B 0,C 180,E1 -20654.4,E2 -20654.4} C_VEL
LIN {X 0,Y 258.804,Z 384.417,A -85,B 0,C 180,E1 -20655.086,E2 -20655.086} C_VEL
LIN {X 0,Y 253.648,Z 372.066,A -85,B 0,C 180,E1 -20656.75,E2 -20656.75} C_VEL
LIN {X 0,Y 247.827,Z 359.773,A -85,B 0,C 180,E1 -20658.708,E2 -20658.708} C_VEL
LIN {X 0,Y 242.023,Z 348.823,A -85,B 0,C 180,E1 -20660.779,E2 -20660.779} C_VEL
LIN {X 0,Y 236.312,Z 338.978,A -85,B 0,C 180,E1 -20662.97,E2 -20662.97} C_VEL
LIN {X 0,Y 230.654,Z 329.858,A -85,B 0,C 180,E1 -20665.337,E2 -20665.337} C_VEL
LIN {X 0,Y 226.407,Z 323.636,A -85,B 0,C 180,E1 -20667.258,E2 -20667.258} C_VEL
LIN {X 0,Y 222.294,Z 317.79,A -85,B 0,C 180,E1 -20669.284,E2 -20669.284} C_VEL
LIN {X 0,Y 219.143,Z 314.128,A -85,B 0,C 180,E1 -20670.922,E2 -20670.922} C_VEL
LIN {X 0,Y 218.184,Z 312.192,A -85,B 0,C 180,E1 -20671.502,E2 -20671.502} C_VEL
LIN {X 0,Y 215.682,Z 310.45,A -85,B 0,C 180,E1 -20672.859,E2 -20672.859} C_VEL
LIN {X 0,Y 214.166,Z 307.946,A -85,B 0,C 180,E1 -20673.835,E2 -20673.835} C_VEL
LIN {X 0,Y 213.804,Z 306.465,A -85,B 0,C 180,E1 -20674.18,E2 -20674.18} C_VEL
LIN {X 0,Y 213.811,Z 306.474,A -85,B 0,C 180,E1 -20678.803,E2 -20678.803} C_VEL
LIN {X 0,Y 213.967,Z 306.459,A -85,B 0,C 180,E1 -20682.806,E2 -20682.806} C_VEL
LIN {X 0,Y 213.958,Z 306.46,A -85,B 0,C 180,E1 -20686.707,E2 -20686.707} C_VEL
LIN {X 0,Y 214.139,Z 306.436,A -85,B 0,C 180,E1 -20690.555,E2 -20690.555} C_VEL
LIN {X 0,Y 214.08,Z 306.438,A -85,B 0,C 180,E1 -20694.348,E2 -20694.348} C_VEL
LIN {X 0,Y 214.411,Z 306.392,A -85,B 0,C 180,E1 -20698.122,E2 -20698.122} C_VEL
LIN {X 0,Y 214.517,Z 306.387,A -85,B 0,C 180,E1 -20700,E2 -20700} C_VEL
LIN {X 0,Y 214.412,Z 306.389,A -85,B 0,C 180,E1 -20701.879,E2 -20701.879} C_VEL
LIN {X 0,Y 214.188,Z 306.425,A -85,B 0,C 180,E1 -20707.542,E2 -20707.542} C_VEL
LIN {X 0,Y 213.988,Z 306.445,A -85,B 0,C 180,E1 -20711.365,E2 -20711.365} C_VEL
LIN {X 0,Y 213.872,Z 306.458,A -85,B 0,C 180,E1 -20715.242,E2 -20715.242} C_VEL
LIN {X 0,Y 213.794,Z 306.468,A -85,B 0,C 180,E1 -20719.192,E2 -20719.192} C_VEL
LIN {X 0,Y 213.792,Z 306.47,A -85,B 0,C 180,E1 -20723.234,E2 -20723.234} C_VEL
LIN {X 0,Y 213.802,Z 306.45,A -85,B 0,C 180,E1 -20726.41,E2 -20726.41} C_VEL
LIN {X 0,Y 214.678,Z 309.127,A -85,B 0,C 180,E1 -20727.105,E2 -20727.105} C_VEL
LIN {X 0,Y 216.531,Z 311.249,A -85,B 0,C 180,E1 -20728.207,E2 -20728.207} C_VEL
LIN {X 0,Y 218.288,Z 312.332,A -85,B 0,C 180,E1 -20729.138,E2 -20729.138} C_VEL
LIN {X 0,Y 220.079,Z 315.496,A -85,B 0,C 180,E1 -20730.177,E2 -20730.177} C_VEL
LIN {X 0,Y 222.664,Z 317.883,A -85,B 0,C 180,E1 -20731.461,E2 -20731.461} C_VEL
LIN {X 0,Y 225.041,Z 321.342,A -85,B 0,C 180,E1 -20732.65,E2 -20732.65} C_VEL
LIN {X 0,Y 226.787,Z 323.241,A -85,B 0,C 180,E1 -20733.448,E2 -20733.448} C_VEL
LIN {X 0,Y 229.716,Z 327.046,A -85,B 0,C 180,E1 -20734.756,E2 -20734.756} C_VEL
LIN {X 0,Y 236.8,Z 336.81,A -85,B 0,C 180,E1 -20737.66,E2 -20737.66} C_VEL
LIN {X 0,Y 244.695,Z 348.604,A -85,B 0,C 180,E1 -20740.545,E2 -20740.545} C_VEL
LIN {X 0,Y 252.25,Z 361.081,A -85,B 0,C 180,E1 -20743.047,E2 -20743.047} C_VEL
LIN {X 0,Y 258.521,Z 372.595,A -85,B 0,C 180,E1 -20744.977,E2 -20744.977} C_VEL
LIN {X 0,Y 259.252,Z 374.317,A -85,B 0,C 180,E1 -20745.206,E2 -20745.206} C_VEL
LIN {X 0,Y 254.28,Z 459.995,A -85,B 0,C 180,E1 -20747.445,E2 -20747.445} C_VEL
LIN {X 0,Y 252.689,Z 474.724,A -85,B 0,C 180,E1 -20748.057,E2 -20748.057} C_VEL
LIN {X 0,Y 250.576,Z 488.649,A -85,B 0,C 180,E1 -20748.9,E2 -20748.9} C_VEL
LIN {X 0,Y 247.689,Z 503.563,A -85,B 0,C 180,E1 -20750.128,E2 -20750.128} C_VEL
LIN {X 0,Y 244.529,Z 516.989,A -85,B 0,C 180,E1 -20751.571,E2 -20751.571} C_VEL
LIN {X 0,Y 240.852,Z 529.733,A -85,B 0,C 180,E1 -20753.259,E2 -20753.259} C_VEL
LIN {X 0,Y 236.591,Z 542.573,A -85,B 0,C 180,E1 -20755.38,E2 -20755.38} C_VEL
LIN {X 0,Y 232.789,Z 552.987,A -85,B 0,C 180,E1 -20757.505,E2 -20757.505} C_VEL
LIN {X 0,Y 228.909,Z 563.205,A -85,B 0,C 180,E1 -20760.071,E2 -20760.071} C_VEL
LIN {X 0,Y 225.372,Z 571.621,A -85,B 0,C 180,E1 -20762.614,E2 -20762.614} C_VEL
LIN {X 0,Y 221.768,Z 579.855,A -85,B 0,C 180,E1 -20765.67,E2 -20765.67} C_VEL
LIN {X 0,Y 218.376,Z 587.581,A -85,B 0,C 180,E1 -20769.266,E2 -20769.266} C_VEL
LIN {X 0,Y 215.784,Z 593.72,A -85,B 0,C 180,E1 -20772.954,E2 -20772.954} C_VEL
LIN {X 0,Y 213.851,Z 598.455,A -85,B 0,C 180,E1 -20776.699,E2 -20776.699} C_VEL
LIN {X 0,Y 212.587,Z 601.915,A -85,B 0,C 180,E1 -20780.485,E2 -20780.485} C_VEL
LIN {X 0,Y 211.932,Z 604.195,A -85,B 0,C 180,E1 -20784.29,E2 -20784.29} C_VEL
LIN {X 0,Y 211.679,Z 605.355,A -85,B 0,C 180,E1 -20788.096,E2 -20788.096} C_VEL
LIN {X 0,Y 211.679,Z 605.367,A -85,B 0,C 180,E1 -20791.902,E2 -20791.902} C_VEL
LIN {X 0,Y 211.972,Z 604.169,A -85,B 0,C 180,E1 -20795.922,E2 -20795.922} C_VEL
LIN {X 0,Y 212.583,Z 602.025,A -85,B 0,C 180,E1 -20799.514,E2 -20799.514} C_VEL
LIN {X 0,Y 213.812,Z 598.608,A -85,B 0,C 180,E1 -20803.301,E2 -20803.301} C_VEL
LIN {X 0,Y 215.734,Z 593.922,A -85,B 0,C 180,E1 -20807.048,E2 -20807.048} C_VEL
LIN {X 0,Y 218.302,Z 587.846,A -85,B 0,C 180,E1 -20810.739,E2 -20810.739} C_VEL
LIN {X 0,Y 221.699,Z 580.182,A -85,B 0,C 180,E1 -20814.337,E2 -20814.337} C_VEL
LIN {X 0,Y 225.274,Z 572.004,A -85,B 0,C 180,E1 -20817.397,E2 -20817.397} C_VEL
LIN {X 0,Y 229.437,Z 562.143,A -85,B 0,C 180,E1 -20820.358,E2 -20820.358} C_VEL
LIN {X 0,Y 232.601,Z 553.697,A -85,B 0,C 180,E1 -20822.464,E2 -20822.464} C_VEL
LIN {X 0,Y 236.883,Z 542.108,A -85,B 0,C 180,E1 -20824.828,E2 -20824.828} C_VEL
LIN {X 0,Y 241.084,Z 529.175,A -85,B 0,C 180,E1 -20826.959,E2 -20826.959} C_VEL
LIN {X 0,Y 244.759,Z 516.316,A -85,B 0,C 180,E1 -20828.647,E2 -20828.647} C_VEL
LIN {X 0,Y 248.139,Z 501.867,A -85,B 0,C 180,E1 -20830.16,E2 -20830.16} C_VEL
LIN {X 0,Y 250.916,Z 487.504,A -85,B 0,C 180,E1 -20831.297,E2 -20831.297} C_VEL
LIN {X 0,Y 253.145,Z 472.195,A -85,B 0,C 180,E1 -20832.183,E2 -20832.183} C_VEL
LIN {X 0,Y 254.53,Z 457.36,A -85,B 0,C 180,E1 -20832.77,E2 -20832.77} C_VEL
LIN {X 0,Y 259.224,Z 377.704,A -85,B 0,C 180,E1 -20834.821,E2 -20834.821} C_VEL
LIN {X 0,Y 259.274,Z 374.079,A -85,B 0,C 180,E1 -20834.949,E2 -20834.949} C_VEL
LIN {X 0,Y 253.011,Z 362.285,A -85,B 0,C 180,E1 -20836.875,E2 -20836.875} C_VEL
LIN {X 0,Y 245.148,Z 349.221,A -85,B 0,C 180,E1 -20839.469,E2 -20839.469} C_VEL
LIN {X 0,Y 238.555,Z 339.297,A -85,B 0,C 180,E1 -20841.849,E2 -20841.849} C_VEL
LIN {X 0,Y 232.347,Z 330.673,A -85,B 0,C 180,E1 -20844.309,E2 -20844.309} C_VEL
LIN {X 0,Y 229.236,Z 326.472,A -85,B 0,C 180,E1 -20845.646,E2 -20845.646} C_VEL
LIN {X 0,Y 226.581,Z 322.82,A -85,B 0,C 180,E1 -20846.858,E2 -20846.858} C_VEL
LIN {X 0,Y 223.637,Z 319.561,A -85,B 0,C 180,E1 -20848.238,E2 -20848.238} C_VEL
LIN {X 0,Y 222.517,Z 317.594,A -85,B 0,C 180,E1 -20848.833,E2 -20848.833} C_VEL
LIN {X 0,Y 219.832,Z 315.18,A -85,B 0,C 180,E1 -20850.178,E2 -20850.178} C_VEL
LIN {X 0,Y 218.252,Z 312.201,A -85,B 0,C 180,E1 -20851.117,E2 -20851.117} C_VEL
LIN {X 0,Y 215.749,Z 310.583,A -85,B 0,C 180,E1 -20852.473,E2 -20852.473} C_VEL
LIN {X 0,Y 214.233,Z 308.158,A -85,B 0,C 180,E1 -20853.45,E2 -20853.45} C_VEL
LIN {X 0,Y 213.763,Z 306.477,A -85,B 0,C 180,E1 -20853.913,E2 -20853.913} C_VEL
LIN {X 0,Y 213.773,Z 306.483,A -85,B 0,C 180,E1 -20858.799,E2 -20858.799} C_VEL
LIN {X 0,Y 213.877,Z 306.463,A -85,B 0,C 180,E1 -20862.798,E2 -20862.798} C_VEL
LIN {X 0,Y 213.914,Z 306.45,A -85,B 0,C 180,E1 -20866.704,E2 -20866.704} C_VEL
LIN {X 0,Y 214.131,Z 306.42,A -85,B 0,C 180,E1 -20870.555,E2 -20870.555} C_VEL
LIN {X 0,Y 214.076,Z 306.437,A -85,B 0,C 180,E1 -20874.348,E2 -20874.348} C_VEL
LIN {X 0,Y 214.407,Z 306.402,A -85,B 0,C 180,E1 -20878.121,E2 -20878.121} C_VEL
LIN {X 0,Y 214.51,Z 306.376,A -85,B 0,C 180,E1 -20880,E2 -20880} C_VEL
LIN {X 0,Y 214.407,Z 306.387,A -85,B 0,C 180,E1 -20881.878,E2 -20881.878} C_VEL
LIN {X 0,Y 214.183,Z 306.423,A -85,B 0,C 180,E1 -20887.542,E2 -20887.542} C_VEL
LIN {X 0,Y 213.997,Z 306.44,A -85,B 0,C 180,E1 -20891.364,E2 -20891.364} C_VEL
LIN {X 0,Y 213.932,Z 306.449,A -85,B 0,C 180,E1 -20895.237,E2 -20895.237} C_VEL
LIN {X 0,Y 213.876,Z 306.46,A -85,B 0,C 180,E1 -20898.692,E2 -20898.692} C_VEL
LIN {X 0,Y 213.515,Z 307.09,A -85,B 0,C 180,E1 -20900.244,E2 -20900.244} C_VEL
LIN {X 0,Y 212.821,Z 308.709,A -85,B 0,C 180,E1 -20901.751,E2 -20901.751} C_VEL
LIN {X 0,Y 212.148,Z 311.806,A -85,B 0,C 180,E1 -20903.693,E2 -20903.693} C_VEL
LIN {X 0,Y 212.712,Z 315.328,A -85,B 0,C 180,E1 -20905.578,E2 -20905.578} C_VEL
LIN {X 0,Y 213.803,Z 317.005,A -85,B 0,C 180,E1 -20906.48,E2 -20906.48} C_VEL
LIN {X 0,Y 216.19,Z 319.164,A -85,B 0,C 180,E1 -20907.86,E2 -20907.86} C_VEL
LIN {X 0,Y 218.47,Z 322.46,A -85,B 0,C 180,E1 -20909.176,E2 -20909.176} C_VEL
LIN {X 0,Y 221.219,Z 325.711,A -85,B 0,C 180,E1 -20910.617,E2 -20910.617} C_VEL
LIN {X 0,Y 226.011,Z 332.978,A -85,B 0,C 180,E1 -20913.008,E2 -20913.008} C_VEL
LIN {X 0,Y 229.402,Z 338.327,A -85,B 0,C 180,E1 -20914.567,E2 -20914.567} C_VEL
LIN {X 0,Y 234.869,Z 347.396,A -85,B 0,C 180,E1 -20916.893,E2 -20916.893} C_VEL
LIN {X 0,Y 241.875,Z 360.277,A -85,B 0,C 180,E1 -20919.62,E2 -20919.62} C_VEL
LIN {X 0,Y 248.179,Z 373.321,A -85,B 0,C 180,E1 -20921.887,E2 -20921.887} C_VEL
LIN {X 0,Y 253.172,Z 385.102,A -85,B 0,C 180,E1 -20923.596,E2 -20923.596} C_VEL
LIN {X 0,Y 253.801,Z 386.776,A -85,B 0,C 180,E1 -20923.81,E2 -20923.81} C_VEL
LIN {X 0,Y 248.457,Z 474.805,A -85,B 0,C 180,E1 -20926.131,E2 -20926.131} C_VEL
LIN {X 0,Y 246.488,Z 490.968,A -85,B 0,C 180,E1 -20926.82,E2 -20926.82} C_VEL
LIN {X 0,Y 243.696,Z 506.225,A -85,B 0,C 180,E1 -20927.755,E2 -20927.755} C_VEL
LIN {X 0,Y 240.513,Z 519.97,A -85,B 0,C 180,E1 -20928.894,E2 -20928.894} C_VEL
LIN {X 0,Y 236.66,Z 534.07,A -85,B 0,C 180,E1 -20930.433,E2 -20930.433} C_VEL
LIN {X 0,Y 232.544,Z 547.173,A -85,B 0,C 180,E1 -20932.267,E2 -20932.267} C_VEL
LIN {X 0,Y 227.992,Z 559.606,A -85,B 0,C 180,E1 -20934.421,E2 -20934.421} C_VEL
LIN {X 0,Y 223.137,Z 571.805,A -85,B 0,C 180,E1 -20937.092,E2 -20937.092} C_VEL
LIN {X 0,Y 218.699,Z 582.45,A -85,B 0,C 180,E1 -20940.04,E2 -20940.04} C_VEL
LIN {X 0,Y 214.738,Z 591.735,A -85,B 0,C 180,E1 -20943.256,E2 -20943.256} C_VEL
LIN {X 0,Y 211.396,Z 599.259,A -85,B 0,C 180,E1 -20946.489,E2 -20946.489} C_VEL
LIN {X 0,Y 208.422,Z 606.289,A -85,B 0,C 180,E1 -20950.295,E2 -20950.295} C_VEL
LIN {X 0,Y 206.343,Z 611.83,A -85,B 0,C 180,E1 -20954.189,E2 -20954.189} C_VEL
LIN {X 0,Y 205.018,Z 616.029,A -85,B 0,C 180,E1 -20958.132,E2 -20958.132} C_VEL
LIN {X 0,Y 204.436,Z 618.985,A -85,B 0,C 180,E1 -20962.097,E2 -20962.097} C_VEL
LIN {X 0,Y 204.364,Z 620.755,A -85,B 0,C 180,E1 -20966.057,E2 -20966.057} C_VEL
LIN {X 0,Y 204.553,Z 621.366,A -85,B 0,C 180,E1 -20970.001,E2 -20970.001} C_VEL
LIN {X 0,Y 204.383,Z 620.653,A -85,B 0,C 180,E1 -20974.288,E2 -20974.288} C_VEL
LIN {X 0,Y 204.435,Z 618.95,A -85,B 0,C 180,E1 -20977.905,E2 -20977.905} C_VEL
LIN {X 0,Y 205.017,Z 615.98,A -85,B 0,C 180,E1 -20981.87,E2 -20981.87} C_VEL
LIN {X 0,Y 206.342,Z 611.768,A -85,B 0,C 180,E1 -20985.813,E2 -20985.813} C_VEL
LIN {X 0,Y 208.422,Z 606.204,A -85,B 0,C 180,E1 -20989.707,E2 -20989.707} C_VEL
LIN {X 0,Y 211.371,Z 599.142,A -85,B 0,C 180,E1 -20993.516,E2 -20993.516} C_VEL
LIN {X 0,Y 214.739,Z 591.606,A -85,B 0,C 180,E1 -20996.745,E2 -20996.745} C_VEL
LIN {X 0,Y 218.546,Z 582.576,A -85,B 0,C 180,E1 -20999.877,E2 -20999.877} C_VEL
LIN {X 0,Y 223.137,Z 571.619,A -85,B 0,C 180,E1 -21002.911,E2 -21002.911} C_VEL
LIN {X 0,Y 227.938,Z 559.369,A -85,B 0,C 180,E1 -21005.59,E2 -21005.59} C_VEL
LIN {X 0,Y 232.539,Z 546.892,A -85,B 0,C 180,E1 -21007.736,E2 -21007.736} C_VEL
LIN {X 0,Y 236.655,Z 533.715,A -85,B 0,C 180,E1 -21009.57,E2 -21009.57} C_VEL
LIN {X 0,Y 240.5,Z 519.512,A -85,B 0,C 180,E1 -21011.111,E2 -21011.111} C_VEL
LIN {X 0,Y 243.681,Z 505.707,A -85,B 0,C 180,E1 -21012.25,E2 -21012.25} C_VEL
LIN {X 0,Y 246.476,Z 490.238,A -85,B 0,C 180,E1 -21013.184,E2 -21013.184} C_VEL
LIN {X 0,Y 248.28,Z 474.906,A -85,B 0,C 180,E1 -21013.84,E2 -21013.84} C_VEL
LIN {X 0,Y 252.753,Z 402.567,A -85,B 0,C 180,E1 -21015.74,E2 -21015.74} C_VEL
LIN {X 0,Y 253.588,Z 386.532,A -85,B 0,C 180,E1 -21016.184,E2 -21016.184} C_VEL
LIN {X 0,Y 248.989,Z 375.386,A -85,B 0,C 180,E1 -21017.751,E2 -21017.751} C_VEL
LIN {X 0,Y 242.977,Z 362.522,A -85,B 0,C 180,E1 -21019.891,E2 -21019.891} C_VEL
LIN {X 0,Y 236.137,Z 349.677,A -85,B 0,C 180,E1 -21022.502,E2 -21022.502} C_VEL
LIN {X 0,Y 230.275,Z 339.74,A -85,B 0,C 180,E1 -21024.947,E2 -21024.947} C_VEL
LIN {X 0,Y 226.876,Z 334.403,A -85,B 0,C 180,E1 -21026.472,E2 -21026.472} C_VEL
LIN {X 0,Y 223.477,Z 329.221,A -85,B 0,C 180,E1 -21028.101,E2 -21028.101} C_VEL
LIN {X 0,Y 219.828,Z 323.897,A -85,B 0,C 180,E1 -21029.981,E2 -21029.981} C_VEL
LIN {X 0,Y 216.693,Z 320.133,A -85,B 0,C 180,E1 -21031.684,E2 -21031.684} C_VEL
LIN {X 0,Y 215.622,Z 318.499,A -85,B 0,C 180,E1 -21032.325,E2 -21032.325} C_VEL
LIN {X 0,Y 213.152,Z 316.256,A -85,B 0,C 180,E1 -21033.767,E2 -21033.767} C_VEL
LIN {X 0,Y 211.477,Z 313.164,A -85,B 0,C 180,E1 -21034.931,E2 -21034.931} C_VEL
LIN {X 0,Y 208.86,Z 311.559,A -85,B 0,C 180,E1 -21036.624,E2 -21036.624} C_VEL
LIN {X 0,Y 207.248,Z 309.225,A -85,B 0,C 180,E1 -21037.869,E2 -21037.869} C_VEL
LIN {X 0,Y 206.761,Z 307.348,A -85,B 0,C 180,E1 -21038.437,E2 -21038.437} C_VEL
LIN {X 0,Y 206.878,Z 307.336,A -85,B 0,C 180,E1 -21042.197,E2 -21042.197} C_VEL
LIN {X 0,Y 206.9,Z 307.335,A -85,B 0,C 180,E1 -21046.245,E2 -21046.245} C_VEL
LIN {X 0,Y 207.083,Z 307.311,A -85,B 0,C 180,E1 -21050.23,E2 -21050.23} C_VEL
LIN {X 0,Y 207.043,Z 307.312,A -85,B 0,C 180,E1 -21054.155,E2 -21054.155} C_VEL
LIN {X 0,Y 207.35,Z 307.271,A -85,B 0,C 180,E1 -21058.058,E2 -21058.058} C_VEL
LIN {X 0,Y 207.485,Z 307.263,A -85,B 0,C 180,E1 -21060,E2 -21060} C_VEL
LIN {X 0,Y 207.352,Z 307.269,A -85,B 0,C 180,E1 -21061.943,E2 -21061.943} C_VEL
LIN {X 0,Y 207.132,Z 307.306,A -85,B 0,C 180,E1 -21067.8,E2 -21067.8} C_VEL
LIN {X 0,Y 206.908,Z 307.33,A -85,B 0,C 180,E1 -21071.76,E2 -21071.76} C_VEL
LIN {X 0,Y 206.806,Z 307.341,A -85,B 0,C 180,E1 -21075.776,E2 -21075.776} C_VEL
LIN {X 0,Y 206.715,Z 307.353,A -85,B 0,C 180,E1 -21079.876,E2 -21079.876} C_VEL
LIN {X 0,Y 206.752,Z 307.539,A -85,B 0,C 180,E1 -21082.223,E2 -21082.223} C_VEL
LIN {X 0,Y 207.508,Z 309.769,A -85,B 0,C 180,E1 -21082.933,E2 -21082.933} C_VEL
LIN {X 0,Y 209.328,Z 312.02,A -85,B 0,C 180,E1 -21084.286,E2 -21084.286} C_VEL
LIN {X 0,Y 211.551,Z 313.365,A -85,B 0,C 180,E1 -21085.708,E2 -21085.708} C_VEL
LIN {X 0,Y 213.164,Z 316.345,A -85,B 0,C 180,E1 -21086.827,E2 -21086.827} C_VEL
LIN {X 0,Y 216.114,Z 319.051,A -85,B 0,C 180,E1 -21088.539,E2 -21088.539} C_VEL
LIN {X 0,Y 218.375,Z 322.414,A -85,B 0,C 180,E1 -21089.845,E2 -21089.845} C_VEL
LIN {X 0,Y 220.38,Z 324.455,A -85,B 0,C 180,E1 -21090.88,E2 -21090.88} C_VEL
LIN {X 0,Y 223.111,Z 328.054,A -85,B 0,C 180,E1 -21092.261,E2 -21092.261} C_VEL
LIN {X 0,Y 224.429,Z 329.775,A -85,B 0,C 180,E1 -21092.897,E2 -21092.897} C_VEL
LIN {X 0,Y 228.33,Z 335.01,A -85,B 0,C 180,E1 -21094.683,E2 -21094.683} C_VEL
LIN {X 0,Y 231.571,Z 339.529,A -85,B 0,C 180,E1 -21096.073,E2 -21096.073} C_VEL
LIN {X 0,Y 238.534,Z 349.678,A -85,B 0,C 180,E1 -21098.815,E2 -21098.815} C_VEL
LIN {X 0,Y 246.487,Z 362.662,A -85,B 0,C 180,E1 -21101.646,E2 -21101.646} C_VEL
LIN {X 0,Y 253.231,Z 375.015,A -85,B 0,C 180,E1 -21103.851,E2 -21103.851} C_VEL
LIN {X 0,Y 254.124,Z 376.747,A -85,B 0,C 180,E1 -21104.132,E2 -21104.132} C_VEL
LIN {X 0,Y 249.119,Z 460.284,A -85,B 0,C 180,E1 -21106.345,E2 -21106.345} C_VEL
LIN {X 0,Y 247.468,Z 475.006,A -85,B 0,C 180,E1 -21106.961,E2 -21106.961} C_VEL
LIN {X 0,Y 245.269,Z 488.928,A -85,B 0,C 180,E1 -21107.809,E2 -21107.809} C_VEL
LIN {X 0,Y 242.497,Z 502.92,A -85,B 0,C 180,E1 -21108.968,E2 -21108.968} C_VEL
LIN {X 0,Y 239.009,Z 517.264,A -85,B 0,C 180,E1 -21110.514,E2 -21110.514} C_VEL
LIN {X 0,Y 235.181,Z 530.009,A -85,B 0,C 180,E1 -21112.22,E2 -21112.22} C_VEL
LIN {X 0,Y 230.794,Z 542.846,A -85,B 0,C 180,E1 -21114.381,E2 -21114.381} C_VEL
LIN {X 0,Y 226.765,Z 553.386,A -85,B 0,C 180,E1 -21116.568,E2 -21116.568} C_VEL
LIN {X 0,Y 222.776,Z 563.478,A -85,B 0,C 180,E1 -21119.159,E2 -21119.159} C_VEL
LIN {X 0,Y 219.079,Z 571.894,A -85,B 0,C 180,E1 -21121.758,E2 -21121.758} C_VEL
LIN {X 0,Y 215.306,Z 580.128,A -85,B 0,C 180,E1 -21124.89,E2 -21124.89} C_VEL
LIN {X 0,Y 211.727,Z 587.854,A -85,B 0,C 180,E1 -21128.583,E2 -21128.583} C_VEL
LIN {X 0,Y 209.004,Z 593.992,A -85,B 0,C 180,E1 -21132.383,E2 -21132.383} C_VEL
LIN {X 0,Y 206.914,Z 598.727,A -85,B 0,C 180,E1 -21136.245,E2 -21136.245} C_VEL
LIN {X 0,Y 205.576,Z 602.187,A -85,B 0,C 180,E1 -21140.157,E2 -21140.157} C_VEL
LIN {X 0,Y 204.848,Z 604.524,A -85,B 0,C 180,E1 -21144.238,E2 -21144.238} C_VEL
LIN {X 0,Y 204.599,Z 605.625,A -85,B 0,C 180,E1 -21148.031,E2 -21148.031} C_VEL
LIN {X 0,Y 204.598,Z 605.637,A -85,B 0,C 180,E1 -21151.968,E2 -21151.968} C_VEL
LIN {X 0,Y 204.867,Z 604.527,A -85,B 0,C 180,E1 -21155.906,E2 -21155.906} C_VEL
LIN {X 0,Y 205.572,Z 602.295,A -85,B 0,C 180,E1 -21159.841,E2 -21159.841} C_VEL
LIN {X 0,Y 206.877,Z 598.879,A -85,B 0,C 180,E1 -21163.756,E2 -21163.756} C_VEL
LIN {X 0,Y 208.949,Z 594.192,A -85,B 0,C 180,E1 -21167.62,E2 -21167.62} C_VEL
LIN {X 0,Y 211.645,Z 588.116,A -85,B 0,C 180,E1 -21171.423,E2 -21171.423} C_VEL
LIN {X 0,Y 215.218,Z 580.452,A -85,B 0,C 180,E1 -21175.119,E2 -21175.119} C_VEL
LIN {X 0,Y 218.975,Z 572.274,A -85,B 0,C 180,E1 -21178.254,E2 -21178.254} C_VEL
LIN {X 0,Y 223.315,Z 562.412,A -85,B 0,C 180,E1 -21181.283,E2 -21181.283} C_VEL
LIN {X 0,Y 227.302,Z 552.304,A -85,B 0,C 180,E1 -21183.816,E2 -21183.816} C_VEL
LIN {X 0,Y 231.893,Z 540.248,A -85,B 0,C 180,E1 -21186.226,E2 -21186.226} C_VEL
LIN {X 0,Y 235.915,Z 528.154,A -85,B 0,C 180,E1 -21188.18,E2 -21188.18} C_VEL
LIN {X 0,Y 239.679,Z 515.007,A -85,B 0,C 180,E1 -21189.898,E2 -21189.898} C_VEL
LIN {X 0,Y 242.984,Z 501.259,A -85,B 0,C 180,E1 -21191.315,E2 -21191.315} C_VEL
LIN {X 0,Y 245.644,Z 487.765,A -85,B 0,C 180,E1 -21192.386,E2 -21192.386} C_VEL
LIN {X 0,Y 247.931,Z 472.453,A -85,B 0,C 180,E1 -21193.285,E2 -21193.285} C_VEL
LIN {X 0,Y 249.373,Z 457.61,A -85,B 0,C 180,E1 -21193.876,E2 -21193.876} C_VEL
LIN {X 0,Y 254.239,Z 377.95,A -85,B 0,C 180,E1 -21195.948,E2 -21195.948} C_VEL
LIN {X 0,Y 254.109,Z 376.595,A -85,B 0,C 180,E1 -21196.033,E2 -21196.033} C_VEL
LIN {X 0,Y 247.567,Z 364.464,A -85,B 0,C 180,E1 -21198.157,E2 -21198.157} C_VEL
LIN {X 0,Y 240.219,Z 352.27,A -85,B 0,C 180,E1 -21200.735,E2 -21200.735} C_VEL
LIN {X 0,Y 233.168,Z 341.589,A -85,B 0,C 180,E1 -21203.466,E2 -21203.466} C_VEL
LIN {X 0,Y 226.548,Z 332.488,A -85,B 0,C 180,E1 -21206.322,E2 -21206.322} C_VEL
LIN {X 0,Y 223.412,Z 328.349,A -85,B 0,C 180,E1 -21207.806,E2 -21207.806} C_VEL
LIN {X 0,Y 220.597,Z 324.802,A -85,B 0,C 180,E1 -21209.22,E2 -21209.22} C_VEL
LIN {X 0,Y 219.765,Z 323.664,A -85,B 0,C 180,E1 -21209.663,E2 -21209.663} C_VEL
LIN {X 0,Y 217.118,Z 320.789,A -85,B 0,C 180,E1 -21211.084,E2 -21211.084} C_VEL
LIN {X 0,Y 215.89,Z 318.662,A -85,B 0,C 180,E1 -21211.834,E2 -21211.834} C_VEL
LIN {X 0,Y 213.33,Z 316.546,A -85,B 0,C 180,E1 -21213.317,E2 -21213.317} C_VEL
LIN {X 0,Y 211.632,Z 313.545,A -85,B 0,C 180,E1 -21214.489,E2 -21214.489} C_VEL
LIN {X 0,Y 208.434,Z 311.175,A -85,B 0,C 180,E1 -21216.624,E2 -21216.624} C_VEL
LIN {X 0,Y 207.024,Z 308.748,A -85,B 0,C 180,E1 -21217.774,E2 -21217.774} C_VEL
LIN {X 0,Y 206.726,Z 307.353,A -85,B 0,C 180,E1 -21218.171,E2 -21218.171} C_VEL
LIN {X 0,Y 206.801,Z 307.338,A -85,B 0,C 180,E1 -21222.19,E2 -21222.19} C_VEL
LIN {X 0,Y 206.855,Z 307.327,A -85,B 0,C 180,E1 -21226.241,E2 -21226.241} C_VEL
LIN {X 0,Y 207.076,Z 307.3,A -85,B 0,C 180,E1 -21230.23,E2 -21230.23} C_VEL
LIN {X 0,Y 207.039,Z 307.315,A -85,B 0,C 180,E1 -21234.155,E2 -21234.155} C_VEL
LIN {X 0,Y 207.347,Z 307.281,A -85,B 0,C 180,E1 -21238.057,E2 -21238.057} C_VEL
LIN {X 0,Y 207.478,Z 307.252,A -85,B 0,C 180,E1 -21240,E2 -21240} C_VEL
LIN {X 0,Y 207.346,Z 307.267,A -85,B 0,C 180,E1 -21241.942,E2 -21241.942} C_VEL
LIN {X 0,Y 207.127,Z 307.305,A -85,B 0,C 180,E1 -21247.8,E2 -21247.8} C_VEL
LIN {X 0,Y 206.923,Z 307.323,A -85,B 0,C 180,E1 -21251.758,E2 -21251.758} C_VEL
LIN {X 0,Y 206.87,Z 307.329,A -85,B 0,C 180,E1 -21255.77,E2 -21255.77} C_VEL
LIN {X 0,Y 206.808,Z 307.339,A -85,B 0,C 180,E1 -21259.866,E2 -21259.866} C_VEL
LIN {X 0,Y 206.785,Z 307.355,A -85,B 0,C 180,E1 -21261.43,E2 -21261.43} C_VEL
LIN {X 0,Y 207.459,Z 309.619,A -85,B 0,C 180,E1 -21262.108,E2 -21262.108} C_VEL
LIN {X 0,Y 209.23,Z 311.867,A -85,B 0,C 180,E1 -21263.448,E2 -21263.448} C_VEL
LIN {X 0,Y 211.602,Z 313.361,A -85,B 0,C 180,E1 -21264.988,E2 -21264.988} C_VEL
LIN {X 0,Y 213.201,Z 316.294,A -85,B 0,C 180,E1 -21266.104,E2 -21266.104} C_VEL
LIN {X 0,Y 213.803,Z 317.005,A -85,B 0,C 180,E1 -21266.48,E2 -21266.48} C_VEL
LIN {X 0,Y 215.041,Z 319.231,A -85,B 0,C 180,E1 -21267.286,E2 -21267.286} C_VEL
LIN {X 0,Y 216.443,Z 324.43,A -85,B 0,C 180,E1 -21268.344,E2 -21268.344} C_VEL
LIN {X 0,Y 217.821,Z 329.873,A -85,B 0,C 180,E1 -21269.36,E2 -21269.36} C_VEL
LIN {X 0,Y 219.076,Z 332.468,A -85,B 0,C 180,E1 -21270.098,E2 -21270.098} C_VEL
LIN {X 0,Y 222.692,Z 337.957,A -85,B 0,C 180,E1 -21271.979,E2 -21271.979} C_VEL
LIN {X 0,Y 226.714,Z 344.438,A -85,B 0,C 180,E1 -21273.917,E2 -21273.917} C_VEL
LIN {X 0,Y 232.807,Z 354.928,A -85,B 0,C 180,E1 -21276.599,E2 -21276.599} C_VEL
LIN {X 0,Y 239.629,Z 368.075,A -85,B 0,C 180,E1 -21279.334,E2 -21279.334} C_VEL
LIN {X 0,Y 245.751,Z 381.572,A -85,B 0,C 180,E1 -21281.612,E2 -21281.612} C_VEL
LIN {X 0,Y 248.764,Z 389.002,A -85,B 0,C 180,E1 -21282.691,E2 -21282.691} C_VEL
LIN {X 0,Y 244.094,Z 465.234,A -85,B 0,C 180,E1 -21284.7,E2 -21284.7} C_VEL
LIN {X 0,Y 242.623,Z 481.452,A -85,B 0,C 180,E1 -21285.232,E2 -21285.232} C_VEL
LIN {X 0,Y 240.471,Z 496.049,A -85,B 0,C 180,E1 -21285.971,E2 -21285.971} C_VEL
LIN {X 0,Y 237.483,Z 510.49,A -85,B 0,C 180,E1 -21286.961,E2 -21286.961} C_VEL
LIN {X 0,Y 234.233,Z 523.272,A -85,B 0,C 180,E1 -21288.119,E2 -21288.119} C_VEL
LIN {X 0,Y 230.282,Z 536.652,A -85,B 0,C 180,E1 -21289.679,E2 -21289.679} C_VEL
LIN {X 0,Y 226.031,Z 549.29,A -85,B 0,C 180,E1 -21291.549,E2 -21291.549} C_VEL
LIN {X 0,Y 221.812,Z 560.349,A -85,B 0,C 180,E1 -21293.554,E2 -21293.554} C_VEL
LIN {X 0,Y 217.155,Z 571.535,A -85,B 0,C 180,E1 -21296.064,E2 -21296.064} C_VEL
LIN {X 0,Y 212.954,Z 581.108,A -85,B 0,C 180,E1 -21298.738,E2 -21298.738} C_VEL
LIN {X 0,Y 208.878,Z 590.241,A -85,B 0,C 180,E1 -21301.898,E2 -21301.898} C_VEL
LIN {X 0,Y 204.829,Z 598.987,A -85,B 0,C 180,E1 -21305.687,E2 -21305.687} C_VEL
LIN {X 0,Y 201.669,Z 606.017,A -85,B 0,C 180,E1 -21309.606,E2 -21309.606} C_VEL
LIN {X 0,Y 199.439,Z 611.557,A -85,B 0,C 180,E1 -21313.627,E2 -21313.627} C_VEL
LIN {X 0,Y 198.007,Z 615.757,A -85,B 0,C 180,E1 -21317.705,E2 -21317.705} C_VEL
LIN {X 0,Y 197.379,Z 618.714,A -85,B 0,C 180,E1 -21321.813,E2 -21321.813} C_VEL
LIN {X 0,Y 197.284,Z 620.485,A -85,B 0,C 180,E1 -21325.915,E2 -21325.915} C_VEL
LIN {X 0,Y 197.468,Z 621.096,A -85,B 0,C 180,E1 -21330.001,E2 -21330.001} C_VEL
LIN {X 0,Y 197.285,Z 620.47,A -85,B 0,C 180,E1 -21334.087,E2 -21334.087} C_VEL
LIN {X 0,Y 197.378,Z 618.678,A -85,B 0,C 180,E1 -21338.189,E2 -21338.189} C_VEL
LIN {X 0,Y 198.005,Z 615.706,A -85,B 0,C 180,E1 -21342.297,E2 -21342.297} C_VEL
LIN {X 0,Y 199.438,Z 611.493,A -85,B 0,C 180,E1 -21346.375,E2 -21346.375} C_VEL
LIN {X 0,Y 201.669,Z 605.929,A -85,B 0,C 180,E1 -21350.396,E2 -21350.396} C_VEL
LIN {X 0,Y 204.799,Z 598.867,A -85,B 0,C 180,E1 -21354.319,E2 -21354.319} C_VEL
LIN {X 0,Y 208.366,Z 591.331,A -85,B 0,C 180,E1 -21357.632,E2 -21357.632} C_VEL
LIN {X 0,Y 212.376,Z 582.249,A -85,B 0,C 180,E1 -21360.859,E2 -21360.859} C_VEL
LIN {X 0,Y 217.15,Z 571.343,A -85,B 0,C 180,E1 -21363.939,E2 -21363.939} C_VEL
LIN {X 0,Y 222.14,Z 559.092,A -85,B 0,C 180,E1 -21366.668,E2 -21366.668} C_VEL
LIN {X 0,Y 226.894,Z 546.752,A -85,B 0,C 180,E1 -21368.818,E2 -21368.818} C_VEL
LIN {X 0,Y 231.207,Z 533.439,A -85,B 0,C 180,E1 -21370.695,E2 -21370.695} C_VEL
LIN {X 0,Y 235.184,Z 519.235,A -85,B 0,C 180,E1 -21372.251,E2 -21372.251} C_VEL
LIN {X 0,Y 238.459,Z 505.428,A -85,B 0,C 180,E1 -21373.401,E2 -21373.401} C_VEL
LIN {X 0,Y 241.338,Z 489.956,A -85,B 0,C 180,E1 -21374.34,E2 -21374.34} C_VEL
LIN {X 0,Y 243.196,Z 474.619,A -85,B 0,C 180,E1 -21375.002,E2 -21375.002} C_VEL
LIN {X 0,Y 247.207,Z 412.472,A -85,B 0,C 180,E1 -21376.651,E2 -21376.651} C_VEL
LIN {X 0,Y 248.622,Z 388.901,A -85,B 0,C 180,E1 -21377.279,E2 -21377.279} C_VEL
LIN {X 0,Y 243.315,Z 376.169,A -85,B 0,C 180,E1 -21379.193,E2 -21379.193} C_VEL
LIN {X 0,Y 237.195,Z 363.351,A -85,B 0,C 180,E1 -21381.522,E2 -21381.522} C_VEL
LIN {X 0,Y 230.312,Z 350.558,A -85,B 0,C 180,E1 -21384.367,E2 -21384.367} C_VEL
LIN {X 0,Y 224.245,Z 340.455,A -85,B 0,C 180,E1 -21387.14,E2 -21387.14} C_VEL
LIN {X 0,Y 220.645,Z 334.896,A -85,B 0,C 180,E1 -21388.939,E2 -21388.939} C_VEL
LIN {X 0,Y 217.249,Z 329.8,A -85,B 0,C 180,E1 -21390.775,E2 -21390.775} C_VEL
LIN {X 0,Y 214.396,Z 326.335,A -85,B 0,C 180,E1 -21392.393,E2 -21392.393} C_VEL
LIN {X 0,Y 213.367,Z 324.891,A -85,B 0,C 180,E1 -21393.023,E2 -21393.023} C_VEL
LIN {X 0,Y 210.762,Z 322.153,A -85,B 0,C 180,E1 -21394.642,E2 -21394.642} C_VEL
LIN {X 0,Y 209.347,Z 319.777,A -85,B 0,C 180,E1 -21395.651,E2 -21395.651} C_VEL
LIN {X 0,Y 206.685,Z 317.649,A -85,B 0,C 180,E1 -21397.499,E2 -21397.499} C_VEL
LIN {X 0,Y 205.009,Z 314.848,A -85,B 0,C 180,E1 -21398.903,E2 -21398.903} C_VEL
LIN {X 0,Y 204.768,Z 314.17,A -85,B 0,C 180,E1 -21399.14,E2 -21399.14} C_VEL
LIN {X 0,Y 202.033,Z 312.589,A -85,B 0,C 180,E1 -21401.415,E2 -21401.415} C_VEL
LIN {X 0,Y 200.286,Z 310.049,A -85,B 0,C 180,E1 -21403.238,E2 -21403.238} C_VEL
LIN {X 0,Y 199.819,Z 308.211,A -85,B 0,C 180,E1 -21403.92,E2 -21403.92} C_VEL
LIN {X 0,Y 200.027,Z 308.186,A -85,B 0,C 180,E1 -21409.882,E2 -21409.882} C_VEL
LIN {X 0,Y 200.007,Z 308.187,A -85,B 0,C 180,E1 -21413.949,E2 -21413.949} C_VEL
LIN {X 0,Y 200.292,Z 308.149,A -85,B 0,C 180,E1 -21417.989,E2 -21417.989} C_VEL
LIN {X 0,Y 200.452,Z 308.139,A -85,B 0,C 180,E1 -21420,E2 -21420} C_VEL
LIN {X 0,Y 200.001,Z 308.198,A -85,B 0,C 180,E1 -21424.03,E2 -21424.03} C_VEL
LIN {X 0,Y 200.08,Z 308.187,A -85,B 0,C 180,E1 -21428.077,E2 -21428.077} C_VEL
LIN {X 0,Y 199.858,Z 308.212,A -85,B 0,C 180,E1 -21432.181,E2 -21432.181} C_VEL
LIN {X 0,Y 199.743,Z 308.313,A -85,B 0,C 180,E1 -21436.612,E2 -21436.612} C_VEL
LIN {X 0,Y 200.385,Z 310.403,A -85,B 0,C 180,E1 -21437.477,E2 -21437.477} C_VEL
LIN {X 0,Y 202.153,Z 312.785,A -85,B 0,C 180,E1 -21439.286,E2 -21439.286} C_VEL
LIN {X 0,Y 204.838,Z 314.386,A -85,B 0,C 180,E1 -21441.512,E2 -21441.512} C_VEL
LIN {X 0,Y 206.447,Z 317.426,A -85,B 0,C 180,E1 -21442.905,E2 -21442.905} C_VEL
LIN {X 0,Y 208.789,Z 319.502,A -85,B 0,C 180,E1 -21444.571,E2 -21444.571} C_VEL
LIN {X 0,Y 209.592,Z 320.097,A -85,B 0,C 180,E1 -21445.101,E2 -21445.101} C_VEL
LIN {X 0,Y 211.597,Z 323.291,A -85,B 0,C 180,E1 -21446.492,E2 -21446.492} C_VEL
LIN {X 0,Y 214.044,Z 325.709,A -85,B 0,C 180,E1 -21447.965,E2 -21447.965} C_VEL
LIN {X 0,Y 216.692,Z 329.286,A -85,B 0,C 180,E1 -21449.51,E2 -21449.51} C_VEL
LIN {X 0,Y 217.956,Z 330.639,A -85,B 0,C 180,E1 -21450.187,E2 -21450.187} C_VEL
LIN {X 0,Y 220.994,Z 334.588,A -85,B 0,C 180,E1 -21451.771,E2 -21451.771} C_VEL
LIN {X 0,Y 226.005,Z 341.539,A -85,B 0,C 180,E1 -21454.178,E2 -21454.178} C_VEL
LIN {X 0,Y 232.766,Z 351.297,A -85,B 0,C 180,E1 -21457.077,E2 -21457.077} C_VEL
LIN {X 0,Y 240.049,Z 363.097,A -85,B 0,C 180,E1 -21459.888,E2 -21459.888} C_VEL
LIN {X 0,Y 246.639,Z 374.761,A -85,B 0,C 180,E1 -21462.205,E2 -21462.205} C_VEL
LIN {X 0,Y 249.135,Z 379.604,A -85,B 0,C 180,E1 -21463.042,E2 -21463.042} C_VEL
LIN {X 0,Y 244.046,Z 460.574,A -85,B 0,C 180,E1 -21465.198,E2 -21465.198} C_VEL
LIN {X 0,Y 242.17,Z 476.204,A -85,B 0,C 180,E1 -21465.852,E2 -21465.852} C_VEL
LIN {X 0,Y 239.625,Z 491.79,A -85,B 0,C 180,E1 -21466.862,E2 -21466.862} C_VEL
LIN {X 0,Y 236.522,Z 506.08,A -85,B 0,C 180,E1 -21468.114,E2 -21468.114} C_VEL
LIN {X 0,Y 232.701,Z 520.664,A -85,B 0,C 180,E1 -21469.791,E2 -21469.791} C_VEL
LIN {X 0,Y 228.359,Z 534.095,A -85,B 0,C 180,E1 -21471.729,E2 -21471.729} C_VEL
LIN {X 0,Y 223.842,Z 546.282,A -85,B 0,C 180,E1 -21473.934,E2 -21473.934} C_VEL
LIN {X 0,Y 219.457,Z 557.082,A -85,B 0,C 180,E1 -21476.371,E2 -21476.371} C_VEL
LIN {X 0,Y 215.32,Z 566.701,A -85,B 0,C 180,E1 -21479.063,E2 -21479.063} C_VEL
LIN {X 0,Y 211.05,Z 575.867,A -85,B 0,C 180,E1 -21482.211,E2 -21482.211} C_VEL
LIN {X 0,Y 207.846,Z 582.483,A -85,B 0,C 180,E1 -21484.996,E2 -21484.996} C_VEL
LIN {X 0,Y 204.295,Z 589.789,A -85,B 0,C 180,E1 -21488.824,E2 -21488.824} C_VEL
LIN {X 0,Y 201.562,Z 595.577,A -85,B 0,C 180,E1 -21492.759,E2 -21492.759} C_VEL
LIN {X 0,Y 200.001,Z 599,A -85,B 0,C 180,E1 -21495.759,E2 -21495.759} C_VEL
LIN {X 0,Y 198.564,Z 602.459,A -85,B 0,C 180,E1 -21499.806,E2 -21499.806} C_VEL
LIN {X 0,Y 197.746,Z 604.917,A -85,B 0,C 180,E1 -21504.347,E2 -21504.347} C_VEL
LIN {X 0,Y 197.52,Z 605.895,A -85,B 0,C 180,E1 -21507.96,E2 -21507.96} C_VEL
LIN {X 0,Y 197.519,Z 605.907,A -85,B 0,C 180,E1 -21512.038,E2 -21512.038} C_VEL
LIN {X 0,Y 197.799,Z 604.798,A -85,B 0,C 180,E1 -21516.118,E2 -21516.118} C_VEL
LIN {X 0,Y 198.559,Z 602.566,A -85,B 0,C 180,E1 -21520.193,E2 -21520.193} C_VEL
LIN {X 0,Y 199.967,Z 599.149,A -85,B 0,C 180,E1 -21524.241,E2 -21524.241} C_VEL
LIN {X 0,Y 202.182,Z 594.462,A -85,B 0,C 180,E1 -21528.23,E2 -21528.23} C_VEL
LIN {X 0,Y 205.21,Z 587.969,A -85,B 0,C 180,E1 -21532.378,E2 -21532.378} C_VEL
LIN {X 0,Y 208.793,Z 580.721,A -85,B 0,C 180,E1 -21535.949,E2 -21535.949} C_VEL
LIN {X 0,Y 212.706,Z 572.544,A -85,B 0,C 180,E1 -21539.166,E2 -21539.166} C_VEL
LIN {X 0,Y 217.226,Z 562.724,A -85,B 0,C 180,E1 -21542.249,E2 -21542.249} C_VEL
LIN {X 0,Y 221.426,Z 552.572,A -85,B 0,C 180,E1 -21544.841,E2 -21544.841} C_VEL
LIN {X 0,Y 226.2,Z 540.515,A -85,B 0,C 180,E1 -21547.29,E2 -21547.29} C_VEL
LIN {X 0,Y 230.387,Z 528.42,A -85,B 0,C 180,E1 -21549.27,E2 -21549.27} C_VEL
LIN {X 0,Y 234.27,Z 515.272,A -85,B 0,C 180,E1 -21551.013,E2 -21551.013} C_VEL
LIN {X 0,Y 237.188,Z 503.598,A -85,B 0,C 180,E1 -21552.257,E2 -21552.257} C_VEL
LIN {X 0,Y 240.225,Z 489.323,A -85,B 0,C 180,E1 -21553.433,E2 -21553.433} C_VEL
LIN {X 0,Y 242.598,Z 474.536,A -85,B 0,C 180,E1 -21554.337,E2 -21554.337} C_VEL
LIN {X 0,Y 244.211,Z 459.362,A -85,B 0,C 180,E1 -21554.98,E2 -21554.98} C_VEL
LIN {X 0,Y 249.217,Z 380.896,A -85,B 0,C 180,E1 -21557.043,E2 -21557.043} C_VEL
LIN {X 0,Y 249.101,Z 379.309,A -85,B 0,C 180,E1 -21557.138,E2 -21557.138} C_VEL
LIN {X 0,Y 242.231,Z 366.697,A -85,B 0,C 180,E1 -21559.499,E2 -21559.499} C_VEL
LIN {X 0,Y 235.473,Z 355.492,A -85,B 0,C 180,E1 -21562.025,E2 -21562.025} C_VEL
LIN {X 0,Y 229.699,Z 346.748,A -85,B 0,C 180,E1 -21564.388,E2 -21564.388} C_VEL
LIN {X 0,Y 223.683,Z 338.236,A -85,B 0,C 180,E1 -21567.114,E2 -21567.114} C_VEL
LIN {X 0,Y 220.569,Z 334.135,A -85,B 0,C 180,E1 -21568.651,E2 -21568.651} C_VEL
LIN {X 0,Y 217.223,Z 329.745,A -85,B 0,C 180,E1 -21570.436,E2 -21570.436} C_VEL
LIN {X 0,Y 214.526,Z 326.516,A -85,B 0,C 180,E1 -21571.971,E2 -21571.971} C_VEL
LIN {X 0,Y 213.571,Z 325.048,A -85,B 0,C 180,E1 -21572.567,E2 -21572.567} C_VEL
LIN {X 0,Y 210.847,Z 322.331,A -85,B 0,C 180,E1 -21574.255,E2 -21574.255} C_VEL
LIN {X 0,Y 209.366,Z 319.813,A -85,B 0,C 180,E1 -21575.323,E2 -21575.323} C_VEL
LIN {X 0,Y 206.669,Z 317.717,A -85,B 0,C 180,E1 -21577.209,E2 -21577.209} C_VEL
LIN {X 0,Y 204.933,Z 314.693,A -85,B 0,C 180,E1 -21578.697,E2 -21578.697} C_VEL
LIN {X 0,Y 204.757,Z 314.165,A -85,B 0,C 180,E1 -21578.875,E2 -21578.875} C_VEL
LIN {X 0,Y 201.974,Z 312.611,A -85,B 0,C 180,E1 -21581.224,E2 -21581.224} C_VEL
LIN {X 0,Y 200.165,Z 309.939,A -85,B 0,C 180,E1 -21583.162,E2 -21583.162} C_VEL
LIN {X 0,Y 199.758,Z 308.227,A -85,B 0,C 180,E1 -21583.849,E2 -21583.849} C_VEL
LIN {X 0,Y 200.021,Z 308.18,A -85,B 0,C 180,E1 -21589.881,E2 -21589.881} C_VEL
LIN {X 0,Y 200.002,Z 308.194,A -85,B 0,C 180,E1 -21593.948,E2 -21593.948} C_VEL
LIN {X 0,Y 200.289,Z 308.158,A -85,B 0,C 180,E1 -21597.989,E2 -21597.989} C_VEL
LIN {X 0,Y 200.446,Z 308.127,A -85,B 0,C 180,E1 -21600,E2 -21600} C_VEL
LIN {X 0,Y 199.994,Z 308.195,A -85,B 0,C 180,E1 -21604.03,E2 -21604.03} C_VEL
LIN {X 0,Y 200.075,Z 308.187,A -85,B 0,C 180,E1 -21608.077,E2 -21608.077} C_VEL
LIN {X 0,Y 199.873,Z 308.205,A -85,B 0,C 180,E1 -21612.179,E2 -21612.179} C_VEL
LIN {X 0,Y 199.836,Z 308.265,A -85,B 0,C 180,E1 -21615.816,E2 -21615.816} C_VEL
LIN {X 0,Y 200.455,Z 310.428,A -85,B 0,C 180,E1 -21616.682,E2 -21616.682} C_VEL
LIN {X 0,Y 202.465,Z 312.923,A -85,B 0,C 180,E1 -21618.729,E2 -21618.729} C_VEL
LIN {X 0,Y 204.853,Z 314.327,A -85,B 0,C 180,E1 -21620.719,E2 -21620.719} C_VEL
LIN {X 0,Y 206.307,Z 317.169,A -85,B 0,C 180,E1 -21622.007,E2 -21622.007} C_VEL
LIN {X 0,Y 208.812,Z 319.468,A -85,B 0,C 180,E1 -21623.821,E2 -21623.821} C_VEL
LIN {X 0,Y 209.68,Z 320.209,A -85,B 0,C 180,E1 -21624.406,E2 -21624.406} C_VEL
LIN {X 0,Y 211.925,Z 323.566,A -85,B 0,C 180,E1 -21625.951,E2 -21625.951} C_VEL
LIN {X 0,Y 214.024,Z 325.608,A -85,B 0,C 180,E1 -21627.217,E2 -21627.217} C_VEL
LIN {X 0,Y 216.583,Z 329.115,A -85,B 0,C 180,E1 -21628.728,E2 -21628.728} C_VEL
LIN {X 0,Y 218.772,Z 331.939,A -85,B 0,C 180,E1 -21629.928,E2 -21629.928} C_VEL
LIN {X 0,Y 219.076,Z 332.468,A -85,B 0,C 180,E1 -21630.098,E2 -21630.098} C_VEL
LIN {X 0,Y 221.018,Z 336.177,A -85,B 0,C 180,E1 -21631.175,E2 -21631.175} C_VEL
LIN {X 0,Y 222.534,Z 340.728,A -85,B 0,C 180,E1 -21632.078,E2 -21632.078} C_VEL
LIN {X 0,Y 225.185,Z 350.632,A -85,B 0,C 180,E1 -21633.688,E2 -21633.688} C_VEL
LIN {X 0,Y 226.87,Z 355.234,A -85,B 0,C 180,E1 -21634.566,E2 -21634.566} C_VEL
LIN {X 0,Y 227.557,Z 356.613,A -85,B 0,C 180,E1 -21634.888,E2 -21634.888} C_VEL
LIN {X 0,Y 234.307,Z 369.625,A -85,B 0,C 180,E1 -21637.808,E2 -21637.808} C_VEL
LIN {X 0,Y 240.156,Z 382.375,A -85,B 0,C 180,E1 -21640.137,E2 -21640.137} C_VEL
LIN {X 0,Y 243.815,Z 391.35,A -85,B 0,C 180,E1 -21641.527,E2 -21641.527} C_VEL
LIN {X 0,Y 239.157,Z 464.985,A -85,B 0,C 180,E1 -21643.492,E2 -21643.492} C_VEL
LIN {X 0,Y 237.634,Z 481.195,A -85,B 0,C 180,E1 -21644.026,E2 -21644.026} C_VEL
LIN {X 0,Y 235.287,Z 496.551,A -85,B 0,C 180,E1 -21644.814,E2 -21644.814} C_VEL
LIN {X 0,Y 232.338,Z 510.226,A -85,B 0,C 180,E1 -21645.765,E2 -21645.765} C_VEL
LIN {X 0,Y 228.989,Z 523.007,A -85,B 0,C 180,E1 -21646.932,E2 -21646.932} C_VEL
LIN {X 0,Y 224.55,Z 537.416,A -85,B 0,C 180,E1 -21648.642,E2 -21648.642} C_VEL
LIN {X 0,Y 220.045,Z 550.2,A -85,B 0,C 180,E1 -21650.597,E2 -21650.597} C_VEL
LIN {X 0,Y 215.26,Z 562.042,A -85,B 0,C 180,E1 -21652.844,E2 -21652.844} C_VEL
LIN {X 0,Y 210.5,Z 572.904,A -85,B 0,C 180,E1 -21655.419,E2 -21655.419} C_VEL
LIN {X 0,Y 206.267,Z 582.131,A -85,B 0,C 180,E1 -21658.123,E2 -21658.123} C_VEL
LIN {X 0,Y 202.014,Z 591.191,A -85,B 0,C 180,E1 -21661.423,E2 -21661.423} C_VEL
LIN {X 0,Y 198.286,Z 598.714,A -85,B 0,C 180,E1 -21664.83,E2 -21664.83} C_VEL
LIN {X 0,Y 194.957,Z 605.744,A -85,B 0,C 180,E1 -21668.871,E2 -21668.871} C_VEL
LIN {X 0,Y 192.567,Z 611.285,A -85,B 0,C 180,E1 -21673.025,E2 -21673.025} C_VEL
LIN {X 0,Y 191.009,Z 615.484,A -85,B 0,C 180,E1 -21677.247,E2 -21677.247} C_VEL
LIN {X 0,Y 190.312,Z 618.442,A -85,B 0,C 180,E1 -21681.506,E2 -21681.506} C_VEL
LIN {X 0,Y 190.19,Z 620.299,A -85,B 0,C 180,E1 -21686.125,E2 -21686.125} C_VEL
LIN {X 0,Y 190.385,Z 620.826,A -85,B 0,C 180,E1 -21690.001,E2 -21690.001} C_VEL
LIN {X 0,Y 190.194,Z 620.199,A -85,B 0,C 180,E1 -21694.239,E2 -21694.239} C_VEL
LIN {X 0,Y 190.311,Z 618.406,A -85,B 0,C 180,E1 -21698.496,E2 -21698.496} C_VEL
LIN {X 0,Y 191.008,Z 615.432,A -85,B 0,C 180,E1 -21702.755,E2 -21702.755} C_VEL
LIN {X 0,Y 192.566,Z 611.219,A -85,B 0,C 180,E1 -21706.977,E2 -21706.977} C_VEL
LIN {X 0,Y 194.957,Z 605.654,A -85,B 0,C 180,E1 -21711.131,E2 -21711.131} C_VEL
LIN {X 0,Y 198.248,Z 598.591,A -85,B 0,C 180,E1 -21715.178,E2 -21715.178} C_VEL
LIN {X 0,Y 202.026,Z 591.055,A -85,B 0,C 180,E1 -21718.577,E2 -21718.577} C_VEL
LIN {X 0,Y 206.259,Z 581.974,A -85,B 0,C 180,E1 -21721.88,E2 -21721.88} C_VEL
LIN {X 0,Y 211.257,Z 571.068,A -85,B 0,C 180,E1 -21725.021,E2 -21725.021} C_VEL
LIN {X 0,Y 216.466,Z 558.817,A -85,B 0,C 180,E1 -21727.794,E2 -21727.794} C_VEL
LIN {X 0,Y 221.295,Z 546.706,A -85,B 0,C 180,E1 -21729.941,E2 -21729.941} C_VEL
LIN {X 0,Y 225.518,Z 534.215,A -85,B 0,C 180,E1 -21731.739,E2 -21731.739} C_VEL
LIN {X 0,Y 229.474,Z 520.802,A -85,B 0,C 180,E1 -21733.258,E2 -21733.258} C_VEL
LIN {X 0,Y 232.825,Z 507.42,A -85,B 0,C 180,E1 -21734.423,E2 -21734.423} C_VEL
LIN {X 0,Y 235.77,Z 492.773,A -85,B 0,C 180,E1 -21735.373,E2 -21735.373} C_VEL
LIN {X 0,Y 237.858,Z 477.809,A -85,B 0,C 180,E1 -21736.073,E2 -21736.073} C_VEL
LIN {X 0,Y 239.612,Z 456.07,A -85,B 0,C 180,E1 -21736.701,E2 -21736.701} C_VEL
LIN {X 0,Y 243.673,Z 391.18,A -85,B 0,C 180,E1 -21738.443,E2 -21738.443} C_VEL
LIN {X 0,Y 237.325,Z 376.106,A -85,B 0,C 180,E1 -21740.883,E2 -21740.883} C_VEL
LIN {X 0,Y 231.373,Z 363.942,A -85,B 0,C 180,E1 -21743.323,E2 -21743.323} C_VEL
LIN {X 0,Y 226.035,Z 354.07,A -85,B 0,C 180,E1 -21745.698,E2 -21745.698} C_VEL
LIN {X 0,Y 221.125,Z 345.734,A -85,B 0,C 180,E1 -21748.083,E2 -21748.083} C_VEL
LIN {X 0,Y 217.383,Z 339.859,A -85,B 0,C 180,E1 -21750.06,E2 -21750.06} C_VEL
LIN {X 0,Y 214.997,Z 336.054,A -85,B 0,C 180,E1 -21751.427,E2 -21751.427} C_VEL
LIN {X 0,Y 212.029,Z 332.332,A -85,B 0,C 180,E1 -21753.187,E2 -21753.187} C_VEL
LIN {X 0,Y 211.059,Z 331.122,A -85,B 0,C 180,E1 -21753.796,E2 -21753.796} C_VEL
LIN {X 0,Y 208.382,Z 327.954,A -85,B 0,C 180,E1 -21755.568,E2 -21755.568} C_VEL
LIN {X 0,Y 207.351,Z 326.303,A -85,B 0,C 180,E1 -21756.331,E2 -21756.331} C_VEL
LIN {X 0,Y 204.851,Z 324.074,A -85,B 0,C 180,E1 -21758.16,E2 -21758.16} C_VEL
LIN {X 0,Y 203.046,Z 320.992,A -85,B 0,C 180,E1 -21759.75,E2 -21759.75} C_VEL
LIN {X 0,Y 200.218,Z 318.928,A -85,B 0,C 180,E1 -21762.265,E2 -21762.265} C_VEL
LIN {X 0,Y 198.515,Z 316.04,A -85,B 0,C 180,E1 -21764.207,E2 -21764.207} C_VEL
LIN {X 0,Y 198.252,Z 315.213,A -85,B 0,C 180,E1 -21764.581,E2 -21764.581} C_VEL
LIN {X 0,Y 194.972,Z 313.281,A -85,B 0,C 180,E1 -21768.829,E2 -21768.829} C_VEL
LIN {X 0,Y 193.179,Z 310.058,A -85,B 0,C 180,E1 -21772.685,E2 -21772.685} C_VEL
LIN {X 0,Y 192.965,Z 309.062,A -85,B 0,C 180,E1 -21773.596,E2 -21773.596} C_VEL
LIN {X 0,Y 193.236,Z 309.027,A -85,B 0,C 180,E1 -21777.916,E2 -21777.916} C_VEL
LIN {X 0,Y 193.419,Z 309.014,A -85,B 0,C 180,E1 -21780,E2 -21780} C_VEL
LIN {X 0,Y 192.948,Z 309.076,A -85,B 0,C 180,E1 -21784.178,E2 -21784.178} C_VEL
LIN {X 0,Y 193.01,Z 309.195,A -85,B 0,C 180,E1 -21787.256,E2 -21787.256} C_VEL
LIN {X 0,Y 194,Z 311.94,A -85,B 0,C 180,E1 -21789.952,E2 -21789.952} C_VEL
LIN {X 0,Y 196.124,Z 314.301,A -85,B 0,C 180,E1 -21793.47,E2 -21793.47} C_VEL
LIN {X 0,Y 198.24,Z 315.408,A -85,B 0,C 180,E1 -21796.014,E2 -21796.014} C_VEL
LIN {X 0,Y 199.656,Z 318.328,A -85,B 0,C 180,E1 -21797.744,E2 -21797.744} C_VEL
